// TIA Portal V20 export
DATA_BLOCK "LPFE_AdditionalAlarmData"   // DB241
TITLE = LPFE_AdditionalAlarmData
{ DB_Accessible_From_OPC_UA := 'FALSE' }
AUTHOR : DI FA SUP
FAMILY : LPFE
// Aditional information required to create the Andon and QAS Digital Events.
// stored: Access Published, DBAccessibleFromOPCUA false, DBAccessibleFromWebserver false, MemoryReserve 100, Namespace PFE
   VAR
      additionalAlarmData { ExternalAccessible := 'False'; ExternalVisible := 'False'; ExternalWritable := 'False'} : Array[0.._.CONFIGURED_ALARMS] of "LPFE_typeAdditionalAlarmData";   // Additional Alarm Data for Digital Events
   END_VAR
BEGIN
   additionalAlarmData[0].AlarmId := 3001;
   additionalAlarmData[1].AlarmId := 4001;
   additionalAlarmData[2].AlarmId := 4002;
   additionalAlarmData[3].AlarmId := 4003;
   additionalAlarmData[4].AlarmId := 4004;
   additionalAlarmData[5].AlarmId := 4006;
   additionalAlarmData[6].AlarmId := 4007;
   additionalAlarmData[7].AlarmId := 4008;
   additionalAlarmData[8].AlarmId := 4009;
   additionalAlarmData[9].AlarmId := 4010;
   additionalAlarmData[10].AlarmId := 4011;
   additionalAlarmData[11].AlarmId := 4012;
   additionalAlarmData[12].AlarmId := 4013;
   additionalAlarmData[13].AlarmId := 4014;
   additionalAlarmData[14].AlarmId := 10001;
   additionalAlarmData[15].AlarmId := 10002;
   additionalAlarmData[16].AlarmId := 10003;
   additionalAlarmData[17].AlarmId := 10004;
   additionalAlarmData[18].AlarmId := 10005;
   additionalAlarmData[19].AlarmId := 10006;
   additionalAlarmData[20].AlarmId := 10007;
   additionalAlarmData[21].AlarmId := 10008;
   additionalAlarmData[22].AlarmId := 11001;
   additionalAlarmData[23].AlarmId := 11002;
   additionalAlarmData[24].AlarmId := 11003;
   additionalAlarmData[25].AlarmId := 11004;
   additionalAlarmData[26].AlarmId := 11005;
   additionalAlarmData[27].AlarmId := 11006;
   additionalAlarmData[28].AlarmId := 11007;
   additionalAlarmData[29].AlarmId := 11008;
   additionalAlarmData[30].AlarmId := 12001;
   additionalAlarmData[31].AlarmId := 12002;
   additionalAlarmData[32].AlarmId := 12003;
   additionalAlarmData[33].AlarmId := 12004;
   additionalAlarmData[34].AlarmId := 12005;
   additionalAlarmData[35].AlarmId := 12006;
   additionalAlarmData[36].AlarmId := 12007;
   additionalAlarmData[37].AlarmId := 12008;
   additionalAlarmData[38].AlarmId := 13001;
   additionalAlarmData[39].AlarmId := 13002;
   additionalAlarmData[40].AlarmId := 13003;
   additionalAlarmData[41].AlarmId := 13004;
   additionalAlarmData[42].AlarmId := 13005;
   additionalAlarmData[43].AlarmId := 13006;
   additionalAlarmData[44].AlarmId := 13007;
   additionalAlarmData[45].AlarmId := 13008;
   additionalAlarmData[46].AlarmId := 20001;
   additionalAlarmData[47].AlarmId := 20002;
   additionalAlarmData[48].AlarmId := 20003;
   additionalAlarmData[49].AlarmId := 20004;
   additionalAlarmData[50].AlarmId := 20005;
   additionalAlarmData[51].AlarmId := 20006;
   additionalAlarmData[52].AlarmId := 20007;
   additionalAlarmData[53].AlarmId := 20008;
   additionalAlarmData[54].AlarmId := 21001;
   additionalAlarmData[55].AlarmId := 21002;
   additionalAlarmData[56].AlarmId := 21003;
   additionalAlarmData[57].AlarmId := 21004;
   additionalAlarmData[58].AlarmId := 21005;
   additionalAlarmData[59].AlarmId := 21006;
   additionalAlarmData[60].AlarmId := 21007;
   additionalAlarmData[61].AlarmId := 21008;
   additionalAlarmData[62].AlarmId := 22001;
   additionalAlarmData[63].AlarmId := 22002;
   additionalAlarmData[64].AlarmId := 22003;
   additionalAlarmData[65].AlarmId := 22004;
   additionalAlarmData[66].AlarmId := 22005;
   additionalAlarmData[67].AlarmId := 22006;
   additionalAlarmData[68].AlarmId := 22007;
   additionalAlarmData[69].AlarmId := 22008;
   additionalAlarmData[70].AlarmId := 23001;
   additionalAlarmData[71].AlarmId := 23002;
   additionalAlarmData[72].AlarmId := 23003;
   additionalAlarmData[73].AlarmId := 23004;
   additionalAlarmData[74].AlarmId := 23005;
   additionalAlarmData[75].AlarmId := 23006;
   additionalAlarmData[76].AlarmId := 23007;
   additionalAlarmData[77].AlarmId := 23008;
   additionalAlarmData[78].AlarmId := 24001;
   additionalAlarmData[79].AlarmId := 24002;
   additionalAlarmData[80].AlarmId := 24003;
   additionalAlarmData[81].AlarmId := 24004;
   additionalAlarmData[82].AlarmId := 24005;
   additionalAlarmData[83].AlarmId := 24006;
   additionalAlarmData[84].AlarmId := 24007;
   additionalAlarmData[85].AlarmId := 24008;
   additionalAlarmData[86].AlarmId := 25001;
   additionalAlarmData[87].AlarmId := 25002;
   additionalAlarmData[88].AlarmId := 25003;
   additionalAlarmData[89].AlarmId := 25004;
   additionalAlarmData[90].AlarmId := 25005;
   additionalAlarmData[91].AlarmId := 25006;
   additionalAlarmData[92].AlarmId := 25007;
   additionalAlarmData[93].AlarmId := 25008;
   additionalAlarmData[94].AlarmId := 26001;
   additionalAlarmData[95].AlarmId := 26002;
   additionalAlarmData[96].AlarmId := 26003;
   additionalAlarmData[97].AlarmId := 26004;
   additionalAlarmData[98].AlarmId := 26005;
   additionalAlarmData[99].AlarmId := 26006;
   additionalAlarmData[100].AlarmId := 26007;
   additionalAlarmData[101].AlarmId := 26008;
   additionalAlarmData[102].AlarmId := 27001;
   additionalAlarmData[103].AlarmId := 27002;
   additionalAlarmData[104].AlarmId := 27003;
   additionalAlarmData[105].AlarmId := 27004;
   additionalAlarmData[106].AlarmId := 27005;
   additionalAlarmData[107].AlarmId := 27006;
   additionalAlarmData[108].AlarmId := 27007;
   additionalAlarmData[109].AlarmId := 27008;
   additionalAlarmData[110].AlarmId := 30001;
   additionalAlarmData[111].AlarmId := 30002;
   additionalAlarmData[112].AlarmId := 30003;
   additionalAlarmData[113].AlarmId := 30004;
   additionalAlarmData[114].AlarmId := 30005;
   additionalAlarmData[115].AlarmId := 30006;
   additionalAlarmData[116].AlarmId := 30007;
   additionalAlarmData[117].AlarmId := 30008;
   additionalAlarmData[118].AlarmId := 30009;
   additionalAlarmData[119].AlarmId := 30010;
   additionalAlarmData[120].AlarmId := 30011;
   additionalAlarmData[121].AlarmId := 31001;
   additionalAlarmData[122].AlarmId := 31002;
   additionalAlarmData[123].AlarmId := 31003;
   additionalAlarmData[124].AlarmId := 31004;
   additionalAlarmData[125].AlarmId := 31005;
   additionalAlarmData[126].AlarmId := 31006;
   additionalAlarmData[127].AlarmId := 31007;
   additionalAlarmData[128].AlarmId := 31008;
   additionalAlarmData[129].AlarmId := 32001;
   additionalAlarmData[130].AlarmId := 32002;
   additionalAlarmData[131].AlarmId := 32003;
   additionalAlarmData[132].AlarmId := 32004;
   additionalAlarmData[133].AlarmId := 32005;
   additionalAlarmData[134].AlarmId := 32006;
   additionalAlarmData[135].AlarmId := 32007;
   additionalAlarmData[136].AlarmId := 32008;
   additionalAlarmData[137].AlarmId := 33001;
   additionalAlarmData[138].AlarmId := 33002;
   additionalAlarmData[139].AlarmId := 33003;
   additionalAlarmData[140].AlarmId := 33004;
   additionalAlarmData[141].AlarmId := 33005;
   additionalAlarmData[142].AlarmId := 33006;
   additionalAlarmData[143].AlarmId := 33007;
   additionalAlarmData[144].AlarmId := 33008;
   additionalAlarmData[145].AlarmId := 34001;
   additionalAlarmData[146].AlarmId := 34002;
   additionalAlarmData[147].AlarmId := 34003;
   additionalAlarmData[148].AlarmId := 34004;
   additionalAlarmData[149].AlarmId := 34005;
   additionalAlarmData[150].AlarmId := 34006;
   additionalAlarmData[151].AlarmId := 34007;
   additionalAlarmData[152].AlarmId := 34008;
   additionalAlarmData[153].AlarmId := 35001;
   additionalAlarmData[154].AlarmId := 35002;
   additionalAlarmData[155].AlarmId := 35003;
   additionalAlarmData[156].AlarmId := 35004;
   additionalAlarmData[157].AlarmId := 35005;
   additionalAlarmData[158].AlarmId := 35006;
   additionalAlarmData[159].AlarmId := 35007;
   additionalAlarmData[160].AlarmId := 35008;
   additionalAlarmData[161].AlarmId := 36001;
   additionalAlarmData[162].AlarmId := 36002;
   additionalAlarmData[163].AlarmId := 36003;
   additionalAlarmData[164].AlarmId := 36004;
   additionalAlarmData[165].AlarmId := 36005;
   additionalAlarmData[166].AlarmId := 36006;
   additionalAlarmData[167].AlarmId := 36007;
   additionalAlarmData[168].AlarmId := 36008;
   additionalAlarmData[169].AlarmId := 40001;
   additionalAlarmData[170].AlarmId := 40002;
   additionalAlarmData[171].AlarmId := 40003;
   additionalAlarmData[172].AlarmId := 40004;
   additionalAlarmData[173].AlarmId := 40005;
   additionalAlarmData[174].AlarmId := 40006;
   additionalAlarmData[175].AlarmId := 40007;
   additionalAlarmData[176].AlarmId := 40008;
   additionalAlarmData[177..999].AlarmId := 0;
   additionalAlarmData[0].priority := 15;
   additionalAlarmData[1..4].priority := 30;
   additionalAlarmData[5].priority := 151;
   additionalAlarmData[6].priority := 104;
   additionalAlarmData[7].priority := 106;
   additionalAlarmData[8].priority := 30;
   additionalAlarmData[9].priority := 151;
   additionalAlarmData[10].priority := 120;
   additionalAlarmData[11].priority := 151;
   additionalAlarmData[12].priority := 105;
   additionalAlarmData[13].priority := 151;
   additionalAlarmData[14].priority := 170;
   additionalAlarmData[15].priority := 106;
   additionalAlarmData[16].priority := 151;
   additionalAlarmData[17].priority := 152;
   additionalAlarmData[18].priority := 170;
   additionalAlarmData[19].priority := 201;
   additionalAlarmData[20].priority := 205;
   additionalAlarmData[21].priority := 251;
   additionalAlarmData[22].priority := 10;
   additionalAlarmData[23].priority := 120;
   additionalAlarmData[24].priority := 151;
   additionalAlarmData[25].priority := 152;
   additionalAlarmData[26].priority := 170;
   additionalAlarmData[27].priority := 204;
   additionalAlarmData[28].priority := 206;
   additionalAlarmData[29].priority := 254;
   additionalAlarmData[30].priority := 15;
   additionalAlarmData[31].priority := 107;
   additionalAlarmData[32].priority := 151;
   additionalAlarmData[33].priority := 152;
   additionalAlarmData[34].priority := 170;
   additionalAlarmData[35].priority := 202;
   additionalAlarmData[36].priority := 205;
   additionalAlarmData[37].priority := 251;
   additionalAlarmData[38].priority := 20;
   additionalAlarmData[39].priority := 105;
   additionalAlarmData[40].priority := 151;
   additionalAlarmData[41].priority := 152;
   additionalAlarmData[42].priority := 170;
   additionalAlarmData[43].priority := 204;
   additionalAlarmData[44].priority := 206;
   additionalAlarmData[45].priority := 251;
   additionalAlarmData[46].priority := 170;
   additionalAlarmData[47].priority := 104;
   additionalAlarmData[48].priority := 151;
   additionalAlarmData[49].priority := 152;
   additionalAlarmData[50].priority := 170;
   additionalAlarmData[51].priority := 202;
   additionalAlarmData[52].priority := 205;
   additionalAlarmData[53].priority := 251;
   additionalAlarmData[54].priority := 35;
   additionalAlarmData[55].priority := 120;
   additionalAlarmData[56].priority := 151;
   additionalAlarmData[57].priority := 152;
   additionalAlarmData[58].priority := 170;
   additionalAlarmData[59].priority := 201;
   additionalAlarmData[60].priority := 206;
   additionalAlarmData[61].priority := 254;
   additionalAlarmData[62].priority := 50;
   additionalAlarmData[63].priority := 105;
   additionalAlarmData[64].priority := 151;
   additionalAlarmData[65].priority := 152;
   additionalAlarmData[66].priority := 170;
   additionalAlarmData[67].priority := 204;
   additionalAlarmData[68].priority := 205;
   additionalAlarmData[69].priority := 254;
   additionalAlarmData[70].priority := 55;
   additionalAlarmData[71].priority := 105;
   additionalAlarmData[72].priority := 151;
   additionalAlarmData[73].priority := 152;
   additionalAlarmData[74].priority := 170;
   additionalAlarmData[75].priority := 202;
   additionalAlarmData[76].priority := 206;
   additionalAlarmData[77].priority := 251;
   additionalAlarmData[78].priority := 60;
   additionalAlarmData[79].priority := 106;
   additionalAlarmData[80].priority := 151;
   additionalAlarmData[81].priority := 152;
   additionalAlarmData[82].priority := 170;
   additionalAlarmData[83].priority := 202;
   additionalAlarmData[84].priority := 206;
   additionalAlarmData[85].priority := 254;
   additionalAlarmData[86].priority := 65;
   additionalAlarmData[87].priority := 104;
   additionalAlarmData[88].priority := 151;
   additionalAlarmData[89].priority := 152;
   additionalAlarmData[90].priority := 170;
   additionalAlarmData[91].priority := 201;
   additionalAlarmData[92].priority := 206;
   additionalAlarmData[93].priority := 251;
   additionalAlarmData[94].priority := 5;
   additionalAlarmData[95].priority := 120;
   additionalAlarmData[96].priority := 151;
   additionalAlarmData[97].priority := 152;
   additionalAlarmData[98].priority := 170;
   additionalAlarmData[99].priority := 201;
   additionalAlarmData[100].priority := 205;
   additionalAlarmData[101].priority := 251;
   additionalAlarmData[102].priority := 10;
   additionalAlarmData[103].priority := 105;
   additionalAlarmData[104].priority := 151;
   additionalAlarmData[105].priority := 152;
   additionalAlarmData[106].priority := 170;
   additionalAlarmData[107].priority := 204;
   additionalAlarmData[108].priority := 206;
   additionalAlarmData[109].priority := 254;
   additionalAlarmData[110].priority := 170;
   additionalAlarmData[111].priority := 106;
   additionalAlarmData[112].priority := 151;
   additionalAlarmData[113].priority := 152;
   additionalAlarmData[114].priority := 170;
   additionalAlarmData[115].priority := 204;
   additionalAlarmData[116].priority := 206;
   additionalAlarmData[117].priority := 251;
   additionalAlarmData[118].priority := 15;
   additionalAlarmData[119].priority := 201;
   additionalAlarmData[120].priority := 251;
   additionalAlarmData[121].priority := 10;
   additionalAlarmData[122].priority := 105;
   additionalAlarmData[123].priority := 151;
   additionalAlarmData[124].priority := 152;
   additionalAlarmData[125].priority := 170;
   additionalAlarmData[126].priority := 204;
   additionalAlarmData[127].priority := 205;
   additionalAlarmData[128].priority := 254;
   additionalAlarmData[129].priority := 35;
   additionalAlarmData[130].priority := 106;
   additionalAlarmData[131].priority := 151;
   additionalAlarmData[132].priority := 152;
   additionalAlarmData[133].priority := 170;
   additionalAlarmData[134].priority := 201;
   additionalAlarmData[135].priority := 205;
   additionalAlarmData[136].priority := 254;
   additionalAlarmData[137].priority := 30;
   additionalAlarmData[138].priority := 105;
   additionalAlarmData[139].priority := 151;
   additionalAlarmData[140].priority := 152;
   additionalAlarmData[141].priority := 170;
   additionalAlarmData[142].priority := 204;
   additionalAlarmData[143].priority := 206;
   additionalAlarmData[144].priority := 251;
   additionalAlarmData[145].priority := 65;
   additionalAlarmData[146].priority := 104;
   additionalAlarmData[147].priority := 151;
   additionalAlarmData[148].priority := 152;
   additionalAlarmData[149].priority := 170;
   additionalAlarmData[150].priority := 201;
   additionalAlarmData[151].priority := 205;
   additionalAlarmData[152].priority := 254;
   additionalAlarmData[153].priority := 60;
   additionalAlarmData[154].priority := 105;
   additionalAlarmData[155].priority := 151;
   additionalAlarmData[156].priority := 152;
   additionalAlarmData[157].priority := 170;
   additionalAlarmData[158].priority := 201;
   additionalAlarmData[159].priority := 206;
   additionalAlarmData[160].priority := 251;
   additionalAlarmData[161].priority := 90;
   additionalAlarmData[162].priority := 120;
   additionalAlarmData[163].priority := 151;
   additionalAlarmData[164].priority := 152;
   additionalAlarmData[165].priority := 170;
   additionalAlarmData[166].priority := 204;
   additionalAlarmData[167].priority := 206;
   additionalAlarmData[168].priority := 254;
   additionalAlarmData[169].priority := 170;
   additionalAlarmData[170].priority := 104;
   additionalAlarmData[171].priority := 151;
   additionalAlarmData[172].priority := 152;
   additionalAlarmData[173].priority := 170;
   additionalAlarmData[174].priority := 204;
   additionalAlarmData[175].priority := 205;
   additionalAlarmData[176].priority := 251;
   additionalAlarmData[177..999].priority := 0;
   additionalAlarmData[0..45].CellID := 1;
   additionalAlarmData[46..109].CellID := 2;
   additionalAlarmData[110..168].CellID := 3;
   additionalAlarmData[169..176].CellID := 4;
   additionalAlarmData[177..999].CellID := 0;
   additionalAlarmData[0].subType := 150;
   additionalAlarmData[1].subType := 0;
   additionalAlarmData[2].subType := 150;
   additionalAlarmData[3].subType := 0;
   additionalAlarmData[4].subType := 150;
   additionalAlarmData[5].subType := 0;
   additionalAlarmData[6].subType := 150;
   additionalAlarmData[7].subType := 0;
   additionalAlarmData[8].subType := 150;
   additionalAlarmData[9].subType := 0;
   additionalAlarmData[10].subType := 150;
   additionalAlarmData[11].subType := 0;
   additionalAlarmData[12].subType := 150;
   additionalAlarmData[13].subType := 0;
   additionalAlarmData[14].subType := 150;
   additionalAlarmData[15].subType := 0;
   additionalAlarmData[16].subType := 150;
   additionalAlarmData[17].subType := 0;
   additionalAlarmData[18].subType := 150;
   additionalAlarmData[19].subType := 0;
   additionalAlarmData[20].subType := 150;
   additionalAlarmData[21].subType := 0;
   additionalAlarmData[22].subType := 150;
   additionalAlarmData[23].subType := 0;
   additionalAlarmData[24].subType := 150;
   additionalAlarmData[25].subType := 0;
   additionalAlarmData[26].subType := 150;
   additionalAlarmData[27].subType := 0;
   additionalAlarmData[28].subType := 150;
   additionalAlarmData[29].subType := 0;
   additionalAlarmData[30].subType := 150;
   additionalAlarmData[31].subType := 0;
   additionalAlarmData[32].subType := 150;
   additionalAlarmData[33].subType := 0;
   additionalAlarmData[34].subType := 150;
   additionalAlarmData[35].subType := 0;
   additionalAlarmData[36].subType := 150;
   additionalAlarmData[37].subType := 0;
   additionalAlarmData[38].subType := 150;
   additionalAlarmData[39].subType := 0;
   additionalAlarmData[40].subType := 150;
   additionalAlarmData[41].subType := 0;
   additionalAlarmData[42].subType := 150;
   additionalAlarmData[43].subType := 0;
   additionalAlarmData[44].subType := 150;
   additionalAlarmData[45].subType := 0;
   additionalAlarmData[46].subType := 150;
   additionalAlarmData[47].subType := 0;
   additionalAlarmData[48].subType := 150;
   additionalAlarmData[49].subType := 0;
   additionalAlarmData[50].subType := 150;
   additionalAlarmData[51].subType := 0;
   additionalAlarmData[52].subType := 150;
   additionalAlarmData[53].subType := 0;
   additionalAlarmData[54].subType := 150;
   additionalAlarmData[55].subType := 0;
   additionalAlarmData[56].subType := 150;
   additionalAlarmData[57].subType := 0;
   additionalAlarmData[58].subType := 150;
   additionalAlarmData[59].subType := 0;
   additionalAlarmData[60].subType := 150;
   additionalAlarmData[61].subType := 0;
   additionalAlarmData[62..63].subType := 150;
   additionalAlarmData[64].subType := 0;
   additionalAlarmData[65].subType := 150;
   additionalAlarmData[66].subType := 0;
   additionalAlarmData[67].subType := 150;
   additionalAlarmData[68].subType := 0;
   additionalAlarmData[69].subType := 150;
   additionalAlarmData[70].subType := 0;
   additionalAlarmData[71].subType := 150;
   additionalAlarmData[72].subType := 0;
   additionalAlarmData[73].subType := 150;
   additionalAlarmData[74].subType := 0;
   additionalAlarmData[75].subType := 150;
   additionalAlarmData[76].subType := 0;
   additionalAlarmData[77].subType := 150;
   additionalAlarmData[78].subType := 0;
   additionalAlarmData[79].subType := 150;
   additionalAlarmData[80].subType := 0;
   additionalAlarmData[81].subType := 150;
   additionalAlarmData[82].subType := 0;
   additionalAlarmData[83].subType := 150;
   additionalAlarmData[84].subType := 0;
   additionalAlarmData[85].subType := 150;
   additionalAlarmData[86].subType := 0;
   additionalAlarmData[87].subType := 150;
   additionalAlarmData[88].subType := 0;
   additionalAlarmData[89].subType := 150;
   additionalAlarmData[90].subType := 0;
   additionalAlarmData[91].subType := 150;
   additionalAlarmData[92].subType := 0;
   additionalAlarmData[93].subType := 150;
   additionalAlarmData[94].subType := 0;
   additionalAlarmData[95].subType := 150;
   additionalAlarmData[96].subType := 0;
   additionalAlarmData[97].subType := 150;
   additionalAlarmData[98].subType := 0;
   additionalAlarmData[99].subType := 150;
   additionalAlarmData[100].subType := 0;
   additionalAlarmData[101].subType := 150;
   additionalAlarmData[102].subType := 0;
   additionalAlarmData[103].subType := 150;
   additionalAlarmData[104].subType := 0;
   additionalAlarmData[105].subType := 150;
   additionalAlarmData[106].subType := 0;
   additionalAlarmData[107].subType := 150;
   additionalAlarmData[108].subType := 0;
   additionalAlarmData[109..110].subType := 150;
   additionalAlarmData[111].subType := 0;
   additionalAlarmData[112].subType := 150;
   additionalAlarmData[113].subType := 0;
   additionalAlarmData[114].subType := 150;
   additionalAlarmData[115].subType := 0;
   additionalAlarmData[116].subType := 150;
   additionalAlarmData[117].subType := 0;
   additionalAlarmData[118..119].subType := 150;
   additionalAlarmData[120].subType := 0;
   additionalAlarmData[121].subType := 150;
   additionalAlarmData[122].subType := 0;
   additionalAlarmData[123].subType := 150;
   additionalAlarmData[124].subType := 0;
   additionalAlarmData[125..126].subType := 150;
   additionalAlarmData[127].subType := 0;
   additionalAlarmData[128].subType := 150;
   additionalAlarmData[129].subType := 0;
   additionalAlarmData[130..131].subType := 150;
   additionalAlarmData[132].subType := 0;
   additionalAlarmData[133].subType := 150;
   additionalAlarmData[134].subType := 0;
   additionalAlarmData[135].subType := 150;
   additionalAlarmData[136].subType := 0;
   additionalAlarmData[137].subType := 150;
   additionalAlarmData[138].subType := 0;
   additionalAlarmData[139].subType := 150;
   additionalAlarmData[140].subType := 0;
   additionalAlarmData[141].subType := 150;
   additionalAlarmData[142].subType := 0;
   additionalAlarmData[143].subType := 150;
   additionalAlarmData[144..145].subType := 0;
   additionalAlarmData[146..148].subType := 150;
   additionalAlarmData[149].subType := 0;
   additionalAlarmData[150].subType := 150;
   additionalAlarmData[151].subType := 0;
   additionalAlarmData[152].subType := 150;
   additionalAlarmData[153].subType := 0;
   additionalAlarmData[154].subType := 150;
   additionalAlarmData[155].subType := 0;
   additionalAlarmData[156].subType := 150;
   additionalAlarmData[157].subType := 0;
   additionalAlarmData[158].subType := 150;
   additionalAlarmData[159].subType := 0;
   additionalAlarmData[160].subType := 150;
   additionalAlarmData[161].subType := 0;
   additionalAlarmData[162].subType := 150;
   additionalAlarmData[163].subType := 0;
   additionalAlarmData[164].subType := 150;
   additionalAlarmData[165..166].subType := 0;
   additionalAlarmData[167].subType := 150;
   additionalAlarmData[168].subType := 0;
   additionalAlarmData[169].subType := 150;
   additionalAlarmData[170].subType := 0;
   additionalAlarmData[171].subType := 150;
   additionalAlarmData[172..173].subType := 0;
   additionalAlarmData[174].subType := 150;
   additionalAlarmData[175].subType := 0;
   additionalAlarmData[176].subType := 150;
   additionalAlarmData[177..999].subType := 0;
   additionalAlarmData[0].classification[0] := 'M';
   additionalAlarmData[0].classification[1] := 'F';
   additionalAlarmData[0].classification[2..3] := ' ';
   additionalAlarmData[1].classification[0] := 'M';
   additionalAlarmData[1].classification[1] := 'F';
   additionalAlarmData[1].classification[2..3] := ' ';
   additionalAlarmData[2].classification[0] := 'M';
   additionalAlarmData[2].classification[1] := 'F';
   additionalAlarmData[2].classification[2..3] := ' ';
   additionalAlarmData[3].classification[0] := 'M';
   additionalAlarmData[3].classification[1] := 'F';
   additionalAlarmData[3].classification[2..3] := ' ';
   additionalAlarmData[4].classification[0] := 'M';
   additionalAlarmData[4].classification[1] := 'F';
   additionalAlarmData[4].classification[2..3] := ' ';
   additionalAlarmData[5].classification[0] := 'T';
   additionalAlarmData[5].classification[1] := 'F';
   additionalAlarmData[5].classification[2] := 'I';
   additionalAlarmData[5].classification[3] := 'B';
   additionalAlarmData[6].classification[0] := 'P';
   additionalAlarmData[6].classification[1] := 'F';
   additionalAlarmData[6].classification[2..3] := ' ';
   additionalAlarmData[7].classification[0] := 'P';
   additionalAlarmData[7].classification[1] := 'F';
   additionalAlarmData[7].classification[2..3] := ' ';
   additionalAlarmData[8].classification[0] := 'M';
   additionalAlarmData[8].classification[1] := 'F';
   additionalAlarmData[8].classification[2..3] := ' ';
   additionalAlarmData[9].classification[0] := 'T';
   additionalAlarmData[9].classification[1] := 'F';
   additionalAlarmData[9].classification[2] := 'I';
   additionalAlarmData[9].classification[3] := 'B';
   additionalAlarmData[10].classification[0] := 'P';
   additionalAlarmData[10].classification[1] := 'F';
   additionalAlarmData[10].classification[2..3] := ' ';
   additionalAlarmData[11].classification[0] := 'T';
   additionalAlarmData[11].classification[1] := 'F';
   additionalAlarmData[11].classification[2] := 'I';
   additionalAlarmData[11].classification[3] := 'B';
   additionalAlarmData[12].classification[0] := 'P';
   additionalAlarmData[12].classification[1] := 'F';
   additionalAlarmData[12].classification[2..3] := ' ';
   additionalAlarmData[13].classification[0] := 'T';
   additionalAlarmData[13].classification[1] := 'F';
   additionalAlarmData[13].classification[2] := 'I';
   additionalAlarmData[13].classification[3] := 'B';
   additionalAlarmData[14].classification[0] := 'S';
   additionalAlarmData[14].classification[1] := 'F';
   additionalAlarmData[14].classification[2..3] := ' ';
   additionalAlarmData[15].classification[0] := 'P';
   additionalAlarmData[15].classification[1] := 'F';
   additionalAlarmData[15].classification[2..3] := ' ';
   additionalAlarmData[16].classification[0] := 'T';
   additionalAlarmData[16].classification[1] := 'F';
   additionalAlarmData[16].classification[2] := 'I';
   additionalAlarmData[16].classification[3] := 'B';
   additionalAlarmData[17].classification[0] := 'T';
   additionalAlarmData[17].classification[1] := 'F';
   additionalAlarmData[17].classification[2] := 'S';
   additionalAlarmData[17].classification[3] := ' ';
   additionalAlarmData[18].classification[0] := 'S';
   additionalAlarmData[18].classification[1] := 'F';
   additionalAlarmData[18].classification[2..3] := ' ';
   additionalAlarmData[19].classification[0] := 'M';
   additionalAlarmData[19].classification[1] := 'W';
   additionalAlarmData[19].classification[2..3] := ' ';
   additionalAlarmData[20].classification[0] := 'P';
   additionalAlarmData[20].classification[1] := 'W';
   additionalAlarmData[20].classification[2..3] := ' ';
   additionalAlarmData[21].classification[0] := 'M';
   additionalAlarmData[21].classification[1] := 'S';
   additionalAlarmData[21].classification[2..3] := ' ';
   additionalAlarmData[22].classification[0] := 'M';
   additionalAlarmData[22].classification[1] := 'F';
   additionalAlarmData[22].classification[2..3] := ' ';
   additionalAlarmData[23].classification[0] := 'P';
   additionalAlarmData[23].classification[1] := 'F';
   additionalAlarmData[23].classification[2..3] := ' ';
   additionalAlarmData[24].classification[0] := 'T';
   additionalAlarmData[24].classification[1] := 'F';
   additionalAlarmData[24].classification[2] := 'I';
   additionalAlarmData[24].classification[3] := 'B';
   additionalAlarmData[25].classification[0] := 'T';
   additionalAlarmData[25].classification[1] := 'F';
   additionalAlarmData[25].classification[2] := 'S';
   additionalAlarmData[25].classification[3] := ' ';
   additionalAlarmData[26].classification[0] := 'S';
   additionalAlarmData[26].classification[1] := 'F';
   additionalAlarmData[26].classification[2..3] := ' ';
   additionalAlarmData[27].classification[0] := 'M';
   additionalAlarmData[27].classification[1] := 'W';
   additionalAlarmData[27].classification[2..3] := ' ';
   additionalAlarmData[28].classification[0] := 'P';
   additionalAlarmData[28].classification[1] := 'W';
   additionalAlarmData[28].classification[2..3] := ' ';
   additionalAlarmData[29].classification[0] := 'M';
   additionalAlarmData[29].classification[1] := 'S';
   additionalAlarmData[29].classification[2..3] := ' ';
   additionalAlarmData[30].classification[0] := 'M';
   additionalAlarmData[30].classification[1] := 'F';
   additionalAlarmData[30].classification[2..3] := ' ';
   additionalAlarmData[31].classification[0] := 'P';
   additionalAlarmData[31].classification[1] := 'F';
   additionalAlarmData[31].classification[2..3] := ' ';
   additionalAlarmData[32].classification[0] := 'T';
   additionalAlarmData[32].classification[1] := 'F';
   additionalAlarmData[32].classification[2] := 'I';
   additionalAlarmData[32].classification[3] := 'B';
   additionalAlarmData[33].classification[0] := 'T';
   additionalAlarmData[33].classification[1] := 'F';
   additionalAlarmData[33].classification[2] := 'S';
   additionalAlarmData[33].classification[3] := ' ';
   additionalAlarmData[34].classification[0] := 'S';
   additionalAlarmData[34].classification[1] := 'F';
   additionalAlarmData[34].classification[2..3] := ' ';
   additionalAlarmData[35].classification[0] := 'M';
   additionalAlarmData[35].classification[1] := 'W';
   additionalAlarmData[35].classification[2..3] := ' ';
   additionalAlarmData[36].classification[0] := 'P';
   additionalAlarmData[36].classification[1] := 'W';
   additionalAlarmData[36].classification[2..3] := ' ';
   additionalAlarmData[37].classification[0] := 'M';
   additionalAlarmData[37].classification[1] := 'S';
   additionalAlarmData[37].classification[2..3] := ' ';
   additionalAlarmData[38].classification[0] := 'M';
   additionalAlarmData[38].classification[1] := 'F';
   additionalAlarmData[38].classification[2..3] := ' ';
   additionalAlarmData[39].classification[0] := 'P';
   additionalAlarmData[39].classification[1] := 'F';
   additionalAlarmData[39].classification[2..3] := ' ';
   additionalAlarmData[40].classification[0] := 'T';
   additionalAlarmData[40].classification[1] := 'F';
   additionalAlarmData[40].classification[2] := 'I';
   additionalAlarmData[40].classification[3] := 'B';
   additionalAlarmData[41].classification[0] := 'T';
   additionalAlarmData[41].classification[1] := 'F';
   additionalAlarmData[41].classification[2] := 'S';
   additionalAlarmData[41].classification[3] := ' ';
   additionalAlarmData[42].classification[0] := 'S';
   additionalAlarmData[42].classification[1] := 'F';
   additionalAlarmData[42].classification[2..3] := ' ';
   additionalAlarmData[43].classification[0] := 'M';
   additionalAlarmData[43].classification[1] := 'W';
   additionalAlarmData[43].classification[2..3] := ' ';
   additionalAlarmData[44].classification[0] := 'P';
   additionalAlarmData[44].classification[1] := 'W';
   additionalAlarmData[44].classification[2..3] := ' ';
   additionalAlarmData[45].classification[0] := 'M';
   additionalAlarmData[45].classification[1] := 'S';
   additionalAlarmData[45].classification[2..3] := ' ';
   additionalAlarmData[46].classification[0] := 'S';
   additionalAlarmData[46].classification[1] := 'F';
   additionalAlarmData[46].classification[2..3] := ' ';
   additionalAlarmData[47].classification[0] := 'P';
   additionalAlarmData[47].classification[1] := 'F';
   additionalAlarmData[47].classification[2..3] := ' ';
   additionalAlarmData[48].classification[0] := 'T';
   additionalAlarmData[48].classification[1] := 'F';
   additionalAlarmData[48].classification[2] := 'I';
   additionalAlarmData[48].classification[3] := 'B';
   additionalAlarmData[49].classification[0] := 'T';
   additionalAlarmData[49].classification[1] := 'F';
   additionalAlarmData[49].classification[2] := 'S';
   additionalAlarmData[49].classification[3] := ' ';
   additionalAlarmData[50].classification[0] := 'S';
   additionalAlarmData[50].classification[1] := 'F';
   additionalAlarmData[50].classification[2..3] := ' ';
   additionalAlarmData[51].classification[0] := 'M';
   additionalAlarmData[51].classification[1] := 'W';
   additionalAlarmData[51].classification[2..3] := ' ';
   additionalAlarmData[52].classification[0] := 'P';
   additionalAlarmData[52].classification[1] := 'W';
   additionalAlarmData[52].classification[2..3] := ' ';
   additionalAlarmData[53].classification[0] := 'M';
   additionalAlarmData[53].classification[1] := 'S';
   additionalAlarmData[53].classification[2..3] := ' ';
   additionalAlarmData[54].classification[0] := 'M';
   additionalAlarmData[54].classification[1] := 'F';
   additionalAlarmData[54].classification[2..3] := ' ';
   additionalAlarmData[55].classification[0] := 'P';
   additionalAlarmData[55].classification[1] := 'F';
   additionalAlarmData[55].classification[2..3] := ' ';
   additionalAlarmData[56].classification[0] := 'T';
   additionalAlarmData[56].classification[1] := 'F';
   additionalAlarmData[56].classification[2] := 'I';
   additionalAlarmData[56].classification[3] := 'B';
   additionalAlarmData[57].classification[0] := 'T';
   additionalAlarmData[57].classification[1] := 'F';
   additionalAlarmData[57].classification[2] := 'S';
   additionalAlarmData[57].classification[3] := ' ';
   additionalAlarmData[58].classification[0] := 'S';
   additionalAlarmData[58].classification[1] := 'F';
   additionalAlarmData[58].classification[2..3] := ' ';
   additionalAlarmData[59].classification[0] := 'M';
   additionalAlarmData[59].classification[1] := 'W';
   additionalAlarmData[59].classification[2..3] := ' ';
   additionalAlarmData[60].classification[0] := 'P';
   additionalAlarmData[60].classification[1] := 'W';
   additionalAlarmData[60].classification[2..3] := ' ';
   additionalAlarmData[61].classification[0] := 'M';
   additionalAlarmData[61].classification[1] := 'S';
   additionalAlarmData[61].classification[2..3] := ' ';
   additionalAlarmData[62].classification[0] := 'M';
   additionalAlarmData[62].classification[1] := 'F';
   additionalAlarmData[62].classification[2..3] := ' ';
   additionalAlarmData[63].classification[0] := 'P';
   additionalAlarmData[63].classification[1] := 'F';
   additionalAlarmData[63].classification[2..3] := ' ';
   additionalAlarmData[64].classification[0] := 'T';
   additionalAlarmData[64].classification[1] := 'F';
   additionalAlarmData[64].classification[2] := 'I';
   additionalAlarmData[64].classification[3] := 'B';
   additionalAlarmData[65].classification[0] := 'T';
   additionalAlarmData[65].classification[1] := 'F';
   additionalAlarmData[65].classification[2] := 'S';
   additionalAlarmData[65].classification[3] := ' ';
   additionalAlarmData[66].classification[0] := 'S';
   additionalAlarmData[66].classification[1] := 'F';
   additionalAlarmData[66].classification[2..3] := ' ';
   additionalAlarmData[67].classification[0] := 'M';
   additionalAlarmData[67].classification[1] := 'W';
   additionalAlarmData[67].classification[2..3] := ' ';
   additionalAlarmData[68].classification[0] := 'P';
   additionalAlarmData[68].classification[1] := 'W';
   additionalAlarmData[68].classification[2..3] := ' ';
   additionalAlarmData[69].classification[0] := 'M';
   additionalAlarmData[69].classification[1] := 'S';
   additionalAlarmData[69].classification[2..3] := ' ';
   additionalAlarmData[70].classification[0] := 'M';
   additionalAlarmData[70].classification[1] := 'F';
   additionalAlarmData[70].classification[2..3] := ' ';
   additionalAlarmData[71].classification[0] := 'P';
   additionalAlarmData[71].classification[1] := 'F';
   additionalAlarmData[71].classification[2..3] := ' ';
   additionalAlarmData[72].classification[0] := 'T';
   additionalAlarmData[72].classification[1] := 'F';
   additionalAlarmData[72].classification[2] := 'I';
   additionalAlarmData[72].classification[3] := 'B';
   additionalAlarmData[73].classification[0] := 'T';
   additionalAlarmData[73].classification[1] := 'F';
   additionalAlarmData[73].classification[2] := 'S';
   additionalAlarmData[73].classification[3] := ' ';
   additionalAlarmData[74].classification[0] := 'S';
   additionalAlarmData[74].classification[1] := 'F';
   additionalAlarmData[74].classification[2..3] := ' ';
   additionalAlarmData[75].classification[0] := 'M';
   additionalAlarmData[75].classification[1] := 'W';
   additionalAlarmData[75].classification[2..3] := ' ';
   additionalAlarmData[76].classification[0] := 'P';
   additionalAlarmData[76].classification[1] := 'W';
   additionalAlarmData[76].classification[2..3] := ' ';
   additionalAlarmData[77].classification[0] := 'M';
   additionalAlarmData[77].classification[1] := 'S';
   additionalAlarmData[77].classification[2..3] := ' ';
   additionalAlarmData[78].classification[0] := 'M';
   additionalAlarmData[78].classification[1] := 'F';
   additionalAlarmData[78].classification[2..3] := ' ';
   additionalAlarmData[79].classification[0] := 'P';
   additionalAlarmData[79].classification[1] := 'F';
   additionalAlarmData[79].classification[2..3] := ' ';
   additionalAlarmData[80].classification[0] := 'T';
   additionalAlarmData[80].classification[1] := 'F';
   additionalAlarmData[80].classification[2] := 'I';
   additionalAlarmData[80].classification[3] := 'B';
   additionalAlarmData[81].classification[0] := 'T';
   additionalAlarmData[81].classification[1] := 'F';
   additionalAlarmData[81].classification[2] := 'S';
   additionalAlarmData[81].classification[3] := ' ';
   additionalAlarmData[82].classification[0] := 'S';
   additionalAlarmData[82].classification[1] := 'F';
   additionalAlarmData[82].classification[2..3] := ' ';
   additionalAlarmData[83].classification[0] := 'M';
   additionalAlarmData[83].classification[1] := 'W';
   additionalAlarmData[83].classification[2..3] := ' ';
   additionalAlarmData[84].classification[0] := 'P';
   additionalAlarmData[84].classification[1] := 'W';
   additionalAlarmData[84].classification[2..3] := ' ';
   additionalAlarmData[85].classification[0] := 'M';
   additionalAlarmData[85].classification[1] := 'S';
   additionalAlarmData[85].classification[2..3] := ' ';
   additionalAlarmData[86].classification[0] := 'M';
   additionalAlarmData[86].classification[1] := 'F';
   additionalAlarmData[86].classification[2..3] := ' ';
   additionalAlarmData[87].classification[0] := 'P';
   additionalAlarmData[87].classification[1] := 'F';
   additionalAlarmData[87].classification[2..3] := ' ';
   additionalAlarmData[88].classification[0] := 'T';
   additionalAlarmData[88].classification[1] := 'F';
   additionalAlarmData[88].classification[2] := 'I';
   additionalAlarmData[88].classification[3] := 'B';
   additionalAlarmData[89].classification[0] := 'T';
   additionalAlarmData[89].classification[1] := 'F';
   additionalAlarmData[89].classification[2] := 'S';
   additionalAlarmData[89].classification[3] := ' ';
   additionalAlarmData[90].classification[0] := 'S';
   additionalAlarmData[90].classification[1] := 'F';
   additionalAlarmData[90].classification[2..3] := ' ';
   additionalAlarmData[91].classification[0] := 'M';
   additionalAlarmData[91].classification[1] := 'W';
   additionalAlarmData[91].classification[2..3] := ' ';
   additionalAlarmData[92].classification[0] := 'P';
   additionalAlarmData[92].classification[1] := 'W';
   additionalAlarmData[92].classification[2..3] := ' ';
   additionalAlarmData[93].classification[0] := 'M';
   additionalAlarmData[93].classification[1] := 'S';
   additionalAlarmData[93].classification[2..3] := ' ';
   additionalAlarmData[94].classification[0] := 'M';
   additionalAlarmData[94].classification[1] := 'F';
   additionalAlarmData[94].classification[2..3] := ' ';
   additionalAlarmData[95].classification[0] := 'P';
   additionalAlarmData[95].classification[1] := 'F';
   additionalAlarmData[95].classification[2..3] := ' ';
   additionalAlarmData[96].classification[0] := 'T';
   additionalAlarmData[96].classification[1] := 'F';
   additionalAlarmData[96].classification[2] := 'I';
   additionalAlarmData[96].classification[3] := 'B';
   additionalAlarmData[97].classification[0] := 'T';
   additionalAlarmData[97].classification[1] := 'F';
   additionalAlarmData[97].classification[2] := 'S';
   additionalAlarmData[97].classification[3] := ' ';
   additionalAlarmData[98].classification[0] := 'S';
   additionalAlarmData[98].classification[1] := 'F';
   additionalAlarmData[98].classification[2..3] := ' ';
   additionalAlarmData[99].classification[0] := 'M';
   additionalAlarmData[99].classification[1] := 'W';
   additionalAlarmData[99].classification[2..3] := ' ';
   additionalAlarmData[100].classification[0] := 'P';
   additionalAlarmData[100].classification[1] := 'W';
   additionalAlarmData[100].classification[2..3] := ' ';
   additionalAlarmData[101].classification[0] := 'M';
   additionalAlarmData[101].classification[1] := 'S';
   additionalAlarmData[101].classification[2..3] := ' ';
   additionalAlarmData[102].classification[0] := 'M';
   additionalAlarmData[102].classification[1] := 'F';
   additionalAlarmData[102].classification[2..3] := ' ';
   additionalAlarmData[103].classification[0] := 'P';
   additionalAlarmData[103].classification[1] := 'F';
   additionalAlarmData[103].classification[2..3] := ' ';
   additionalAlarmData[104].classification[0] := 'T';
   additionalAlarmData[104].classification[1] := 'F';
   additionalAlarmData[104].classification[2] := 'I';
   additionalAlarmData[104].classification[3] := 'B';
   additionalAlarmData[105].classification[0] := 'T';
   additionalAlarmData[105].classification[1] := 'F';
   additionalAlarmData[105].classification[2] := 'S';
   additionalAlarmData[105].classification[3] := ' ';
   additionalAlarmData[106].classification[0] := 'S';
   additionalAlarmData[106].classification[1] := 'F';
   additionalAlarmData[106].classification[2..3] := ' ';
   additionalAlarmData[107].classification[0] := 'M';
   additionalAlarmData[107].classification[1] := 'W';
   additionalAlarmData[107].classification[2..3] := ' ';
   additionalAlarmData[108].classification[0] := 'P';
   additionalAlarmData[108].classification[1] := 'W';
   additionalAlarmData[108].classification[2..3] := ' ';
   additionalAlarmData[109].classification[0] := 'M';
   additionalAlarmData[109].classification[1] := 'S';
   additionalAlarmData[109].classification[2..3] := ' ';
   additionalAlarmData[110].classification[0] := 'S';
   additionalAlarmData[110].classification[1] := 'F';
   additionalAlarmData[110].classification[2..3] := ' ';
   additionalAlarmData[111].classification[0] := 'P';
   additionalAlarmData[111].classification[1] := 'F';
   additionalAlarmData[111].classification[2..3] := ' ';
   additionalAlarmData[112].classification[0] := 'T';
   additionalAlarmData[112].classification[1] := 'F';
   additionalAlarmData[112].classification[2] := 'I';
   additionalAlarmData[112].classification[3] := 'B';
   additionalAlarmData[113].classification[0] := 'T';
   additionalAlarmData[113].classification[1] := 'F';
   additionalAlarmData[113].classification[2] := 'S';
   additionalAlarmData[113].classification[3] := ' ';
   additionalAlarmData[114].classification[0] := 'S';
   additionalAlarmData[114].classification[1] := 'F';
   additionalAlarmData[114].classification[2..3] := ' ';
   additionalAlarmData[115].classification[0] := 'M';
   additionalAlarmData[115].classification[1] := 'W';
   additionalAlarmData[115].classification[2..3] := ' ';
   additionalAlarmData[116].classification[0] := 'P';
   additionalAlarmData[116].classification[1] := 'W';
   additionalAlarmData[116].classification[2..3] := ' ';
   additionalAlarmData[117].classification[0] := 'M';
   additionalAlarmData[117].classification[1] := 'S';
   additionalAlarmData[117].classification[2..3] := ' ';
   additionalAlarmData[118].classification[0] := 'M';
   additionalAlarmData[118].classification[1] := 'F';
   additionalAlarmData[118].classification[2..3] := ' ';
   additionalAlarmData[119].classification[0] := 'M';
   additionalAlarmData[119].classification[1] := 'W';
   additionalAlarmData[119].classification[2..3] := ' ';
   additionalAlarmData[120].classification[0] := 'M';
   additionalAlarmData[120].classification[1] := 'S';
   additionalAlarmData[120].classification[2..3] := ' ';
   additionalAlarmData[121].classification[0] := 'M';
   additionalAlarmData[121].classification[1] := 'F';
   additionalAlarmData[121].classification[2..3] := ' ';
   additionalAlarmData[122].classification[0] := 'P';
   additionalAlarmData[122].classification[1] := 'F';
   additionalAlarmData[122].classification[2..3] := ' ';
   additionalAlarmData[123].classification[0] := 'T';
   additionalAlarmData[123].classification[1] := 'F';
   additionalAlarmData[123].classification[2] := 'I';
   additionalAlarmData[123].classification[3] := 'B';
   additionalAlarmData[124].classification[0] := 'T';
   additionalAlarmData[124].classification[1] := 'F';
   additionalAlarmData[124].classification[2] := 'S';
   additionalAlarmData[124].classification[3] := ' ';
   additionalAlarmData[125].classification[0] := 'S';
   additionalAlarmData[125].classification[1] := 'F';
   additionalAlarmData[125].classification[2..3] := ' ';
   additionalAlarmData[126].classification[0] := 'M';
   additionalAlarmData[126].classification[1] := 'W';
   additionalAlarmData[126].classification[2..3] := ' ';
   additionalAlarmData[127].classification[0] := 'P';
   additionalAlarmData[127].classification[1] := 'W';
   additionalAlarmData[127].classification[2..3] := ' ';
   additionalAlarmData[128].classification[0] := 'M';
   additionalAlarmData[128].classification[1] := 'S';
   additionalAlarmData[128].classification[2..3] := ' ';
   additionalAlarmData[129].classification[0] := 'M';
   additionalAlarmData[129].classification[1] := 'F';
   additionalAlarmData[129].classification[2..3] := ' ';
   additionalAlarmData[130].classification[0] := 'P';
   additionalAlarmData[130].classification[1] := 'F';
   additionalAlarmData[130].classification[2..3] := ' ';
   additionalAlarmData[131].classification[0] := 'T';
   additionalAlarmData[131].classification[1] := 'F';
   additionalAlarmData[131].classification[2] := 'I';
   additionalAlarmData[131].classification[3] := 'B';
   additionalAlarmData[132].classification[0] := 'T';
   additionalAlarmData[132].classification[1] := 'F';
   additionalAlarmData[132].classification[2] := 'S';
   additionalAlarmData[132].classification[3] := ' ';
   additionalAlarmData[133].classification[0] := 'S';
   additionalAlarmData[133].classification[1] := 'F';
   additionalAlarmData[133].classification[2..3] := ' ';
   additionalAlarmData[134].classification[0] := 'M';
   additionalAlarmData[134].classification[1] := 'W';
   additionalAlarmData[134].classification[2..3] := ' ';
   additionalAlarmData[135].classification[0] := 'P';
   additionalAlarmData[135].classification[1] := 'W';
   additionalAlarmData[135].classification[2..3] := ' ';
   additionalAlarmData[136].classification[0] := 'M';
   additionalAlarmData[136].classification[1] := 'S';
   additionalAlarmData[136].classification[2..3] := ' ';
   additionalAlarmData[137].classification[0] := 'M';
   additionalAlarmData[137].classification[1] := 'F';
   additionalAlarmData[137].classification[2..3] := ' ';
   additionalAlarmData[138].classification[0] := 'P';
   additionalAlarmData[138].classification[1] := 'F';
   additionalAlarmData[138].classification[2..3] := ' ';
   additionalAlarmData[139].classification[0] := 'T';
   additionalAlarmData[139].classification[1] := 'F';
   additionalAlarmData[139].classification[2] := 'I';
   additionalAlarmData[139].classification[3] := 'B';
   additionalAlarmData[140].classification[0] := 'T';
   additionalAlarmData[140].classification[1] := 'F';
   additionalAlarmData[140].classification[2] := 'S';
   additionalAlarmData[140].classification[3] := ' ';
   additionalAlarmData[141].classification[0] := 'S';
   additionalAlarmData[141].classification[1] := 'F';
   additionalAlarmData[141].classification[2..3] := ' ';
   additionalAlarmData[142].classification[0] := 'M';
   additionalAlarmData[142].classification[1] := 'W';
   additionalAlarmData[142].classification[2..3] := ' ';
   additionalAlarmData[143].classification[0] := 'P';
   additionalAlarmData[143].classification[1] := 'W';
   additionalAlarmData[143].classification[2..3] := ' ';
   additionalAlarmData[144].classification[0] := 'M';
   additionalAlarmData[144].classification[1] := 'S';
   additionalAlarmData[144].classification[2..3] := ' ';
   additionalAlarmData[145].classification[0] := 'M';
   additionalAlarmData[145].classification[1] := 'F';
   additionalAlarmData[145].classification[2..3] := ' ';
   additionalAlarmData[146].classification[0] := 'P';
   additionalAlarmData[146].classification[1] := 'F';
   additionalAlarmData[146].classification[2..3] := ' ';
   additionalAlarmData[147].classification[0] := 'T';
   additionalAlarmData[147].classification[1] := 'F';
   additionalAlarmData[147].classification[2] := 'I';
   additionalAlarmData[147].classification[3] := 'B';
   additionalAlarmData[148].classification[0] := 'T';
   additionalAlarmData[148].classification[1] := 'F';
   additionalAlarmData[148].classification[2] := 'S';
   additionalAlarmData[148].classification[3] := ' ';
   additionalAlarmData[149].classification[0] := 'S';
   additionalAlarmData[149].classification[1] := 'F';
   additionalAlarmData[149].classification[2..3] := ' ';
   additionalAlarmData[150].classification[0] := 'M';
   additionalAlarmData[150].classification[1] := 'W';
   additionalAlarmData[150].classification[2..3] := ' ';
   additionalAlarmData[151].classification[0] := 'P';
   additionalAlarmData[151].classification[1] := 'W';
   additionalAlarmData[151].classification[2..3] := ' ';
   additionalAlarmData[152].classification[0] := 'M';
   additionalAlarmData[152].classification[1] := 'S';
   additionalAlarmData[152].classification[2..3] := ' ';
   additionalAlarmData[153].classification[0] := 'M';
   additionalAlarmData[153].classification[1] := 'F';
   additionalAlarmData[153].classification[2..3] := ' ';
   additionalAlarmData[154].classification[0] := 'P';
   additionalAlarmData[154].classification[1] := 'F';
   additionalAlarmData[154].classification[2..3] := ' ';
   additionalAlarmData[155].classification[0] := 'T';
   additionalAlarmData[155].classification[1] := 'F';
   additionalAlarmData[155].classification[2] := 'I';
   additionalAlarmData[155].classification[3] := 'B';
   additionalAlarmData[156].classification[0] := 'T';
   additionalAlarmData[156].classification[1] := 'F';
   additionalAlarmData[156].classification[2] := 'S';
   additionalAlarmData[156].classification[3] := ' ';
   additionalAlarmData[157].classification[0] := 'S';
   additionalAlarmData[157].classification[1] := 'F';
   additionalAlarmData[157].classification[2..3] := ' ';
   additionalAlarmData[158].classification[0] := 'M';
   additionalAlarmData[158].classification[1] := 'W';
   additionalAlarmData[158].classification[2..3] := ' ';
   additionalAlarmData[159].classification[0] := 'P';
   additionalAlarmData[159].classification[1] := 'W';
   additionalAlarmData[159].classification[2..3] := ' ';
   additionalAlarmData[160].classification[0] := 'M';
   additionalAlarmData[160].classification[1] := 'S';
   additionalAlarmData[160].classification[2..3] := ' ';
   additionalAlarmData[161].classification[0] := 'M';
   additionalAlarmData[161].classification[1] := 'F';
   additionalAlarmData[161].classification[2..3] := ' ';
   additionalAlarmData[162].classification[0] := 'P';
   additionalAlarmData[162].classification[1] := 'F';
   additionalAlarmData[162].classification[2..3] := ' ';
   additionalAlarmData[163].classification[0] := 'T';
   additionalAlarmData[163].classification[1] := 'F';
   additionalAlarmData[163].classification[2] := 'I';
   additionalAlarmData[163].classification[3] := 'B';
   additionalAlarmData[164].classification[0] := 'T';
   additionalAlarmData[164].classification[1] := 'F';
   additionalAlarmData[164].classification[2] := 'S';
   additionalAlarmData[164].classification[3] := ' ';
   additionalAlarmData[165].classification[0] := 'S';
   additionalAlarmData[165].classification[1] := 'F';
   additionalAlarmData[165].classification[2..3] := ' ';
   additionalAlarmData[166].classification[0] := 'M';
   additionalAlarmData[166].classification[1] := 'W';
   additionalAlarmData[166].classification[2..3] := ' ';
   additionalAlarmData[167].classification[0] := 'P';
   additionalAlarmData[167].classification[1] := 'W';
   additionalAlarmData[167].classification[2..3] := ' ';
   additionalAlarmData[168].classification[0] := 'M';
   additionalAlarmData[168].classification[1] := 'S';
   additionalAlarmData[168].classification[2..3] := ' ';
   additionalAlarmData[169].classification[0] := 'S';
   additionalAlarmData[169].classification[1] := 'F';
   additionalAlarmData[169].classification[2..3] := ' ';
   additionalAlarmData[170].classification[0] := 'P';
   additionalAlarmData[170].classification[1] := 'F';
   additionalAlarmData[170].classification[2..3] := ' ';
   additionalAlarmData[171].classification[0] := 'T';
   additionalAlarmData[171].classification[1] := 'F';
   additionalAlarmData[171].classification[2] := 'I';
   additionalAlarmData[171].classification[3] := 'B';
   additionalAlarmData[172].classification[0] := 'T';
   additionalAlarmData[172].classification[1] := 'F';
   additionalAlarmData[172].classification[2] := 'S';
   additionalAlarmData[172].classification[3] := ' ';
   additionalAlarmData[173].classification[0] := 'S';
   additionalAlarmData[173].classification[1] := 'F';
   additionalAlarmData[173].classification[2..3] := ' ';
   additionalAlarmData[174].classification[0] := 'M';
   additionalAlarmData[174].classification[1] := 'W';
   additionalAlarmData[174].classification[2..3] := ' ';
   additionalAlarmData[175].classification[0] := 'P';
   additionalAlarmData[175].classification[1] := 'W';
   additionalAlarmData[175].classification[2..3] := ' ';
   additionalAlarmData[176].classification[0] := 'M';
   additionalAlarmData[176].classification[1] := 'S';
   additionalAlarmData[176].classification[2..3] := ' ';
   additionalAlarmData[177].classification[0..3] := ' ';
   additionalAlarmData[178].classification[0..3] := ' ';
   additionalAlarmData[179].classification[0..3] := ' ';
   additionalAlarmData[180].classification[0..3] := ' ';
   additionalAlarmData[181].classification[0..3] := ' ';
   additionalAlarmData[182].classification[0..3] := ' ';
   additionalAlarmData[183].classification[0..3] := ' ';
   additionalAlarmData[184].classification[0..3] := ' ';
   additionalAlarmData[185].classification[0..3] := ' ';
   additionalAlarmData[186].classification[0..3] := ' ';
   additionalAlarmData[187].classification[0..3] := ' ';
   additionalAlarmData[188].classification[0..3] := ' ';
   additionalAlarmData[189].classification[0..3] := ' ';
   additionalAlarmData[190].classification[0..3] := ' ';
   additionalAlarmData[191].classification[0..3] := ' ';
   additionalAlarmData[192].classification[0..3] := ' ';
   additionalAlarmData[193].classification[0..3] := ' ';
   additionalAlarmData[194].classification[0..3] := ' ';
   additionalAlarmData[195].classification[0..3] := ' ';
   additionalAlarmData[196].classification[0..3] := ' ';
   additionalAlarmData[197].classification[0..3] := ' ';
   additionalAlarmData[198].classification[0..3] := ' ';
   additionalAlarmData[199].classification[0..3] := ' ';
   additionalAlarmData[200].classification[0..3] := ' ';
   additionalAlarmData[201].classification[0..3] := ' ';
   additionalAlarmData[202].classification[0..3] := ' ';
   additionalAlarmData[203].classification[0..3] := ' ';
   additionalAlarmData[204].classification[0..3] := ' ';
   additionalAlarmData[205].classification[0..3] := ' ';
   additionalAlarmData[206].classification[0..3] := ' ';
   additionalAlarmData[207].classification[0..3] := ' ';
   additionalAlarmData[208].classification[0..3] := ' ';
   additionalAlarmData[209].classification[0..3] := ' ';
   additionalAlarmData[210].classification[0..3] := ' ';
   additionalAlarmData[211].classification[0..3] := ' ';
   additionalAlarmData[212].classification[0..3] := ' ';
   additionalAlarmData[213].classification[0..3] := ' ';
   additionalAlarmData[214].classification[0..3] := ' ';
   additionalAlarmData[215].classification[0..3] := ' ';
   additionalAlarmData[216].classification[0..3] := ' ';
   additionalAlarmData[217].classification[0..3] := ' ';
   additionalAlarmData[218].classification[0..3] := ' ';
   additionalAlarmData[219].classification[0..3] := ' ';
   additionalAlarmData[220].classification[0..3] := ' ';
   additionalAlarmData[221].classification[0..3] := ' ';
   additionalAlarmData[222].classification[0..3] := ' ';
   additionalAlarmData[223].classification[0..3] := ' ';
   additionalAlarmData[224].classification[0..3] := ' ';
   additionalAlarmData[225].classification[0..3] := ' ';
   additionalAlarmData[226].classification[0..3] := ' ';
   additionalAlarmData[227].classification[0..3] := ' ';
   additionalAlarmData[228].classification[0..3] := ' ';
   additionalAlarmData[229].classification[0..3] := ' ';
   additionalAlarmData[230].classification[0..3] := ' ';
   additionalAlarmData[231].classification[0..3] := ' ';
   additionalAlarmData[232].classification[0..3] := ' ';
   additionalAlarmData[233].classification[0..3] := ' ';
   additionalAlarmData[234].classification[0..3] := ' ';
   additionalAlarmData[235].classification[0..3] := ' ';
   additionalAlarmData[236].classification[0..3] := ' ';
   additionalAlarmData[237].classification[0..3] := ' ';
   additionalAlarmData[238].classification[0..3] := ' ';
   additionalAlarmData[239].classification[0..3] := ' ';
   additionalAlarmData[240].classification[0..3] := ' ';
   additionalAlarmData[241].classification[0..3] := ' ';
   additionalAlarmData[242].classification[0..3] := ' ';
   additionalAlarmData[243].classification[0..3] := ' ';
   additionalAlarmData[244].classification[0..3] := ' ';
   additionalAlarmData[245].classification[0..3] := ' ';
   additionalAlarmData[246].classification[0..3] := ' ';
   additionalAlarmData[247].classification[0..3] := ' ';
   additionalAlarmData[248].classification[0..3] := ' ';
   additionalAlarmData[249].classification[0..3] := ' ';
   additionalAlarmData[250].classification[0..3] := ' ';
   additionalAlarmData[251].classification[0..3] := ' ';
   additionalAlarmData[252].classification[0..3] := ' ';
   additionalAlarmData[253].classification[0..3] := ' ';
   additionalAlarmData[254].classification[0..3] := ' ';
   additionalAlarmData[255].classification[0..3] := ' ';
   additionalAlarmData[256].classification[0..3] := ' ';
   additionalAlarmData[257].classification[0..3] := ' ';
   additionalAlarmData[258].classification[0..3] := ' ';
   additionalAlarmData[259].classification[0..3] := ' ';
   additionalAlarmData[260].classification[0..3] := ' ';
   additionalAlarmData[261].classification[0..3] := ' ';
   additionalAlarmData[262].classification[0..3] := ' ';
   additionalAlarmData[263].classification[0..3] := ' ';
   additionalAlarmData[264].classification[0..3] := ' ';
   additionalAlarmData[265].classification[0..3] := ' ';
   additionalAlarmData[266].classification[0..3] := ' ';
   additionalAlarmData[267].classification[0..3] := ' ';
   additionalAlarmData[268].classification[0..3] := ' ';
   additionalAlarmData[269].classification[0..3] := ' ';
   additionalAlarmData[270].classification[0..3] := ' ';
   additionalAlarmData[271].classification[0..3] := ' ';
   additionalAlarmData[272].classification[0..3] := ' ';
   additionalAlarmData[273].classification[0..3] := ' ';
   additionalAlarmData[274].classification[0..3] := ' ';
   additionalAlarmData[275].classification[0..3] := ' ';
   additionalAlarmData[276].classification[0..3] := ' ';
   additionalAlarmData[277].classification[0..3] := ' ';
   additionalAlarmData[278].classification[0..3] := ' ';
   additionalAlarmData[279].classification[0..3] := ' ';
   additionalAlarmData[280].classification[0..3] := ' ';
   additionalAlarmData[281].classification[0..3] := ' ';
   additionalAlarmData[282].classification[0..3] := ' ';
   additionalAlarmData[283].classification[0..3] := ' ';
   additionalAlarmData[284].classification[0..3] := ' ';
   additionalAlarmData[285].classification[0..3] := ' ';
   additionalAlarmData[286].classification[0..3] := ' ';
   additionalAlarmData[287].classification[0..3] := ' ';
   additionalAlarmData[288].classification[0..3] := ' ';
   additionalAlarmData[289].classification[0..3] := ' ';
   additionalAlarmData[290].classification[0..3] := ' ';
   additionalAlarmData[291].classification[0..3] := ' ';
   additionalAlarmData[292].classification[0..3] := ' ';
   additionalAlarmData[293].classification[0..3] := ' ';
   additionalAlarmData[294].classification[0..3] := ' ';
   additionalAlarmData[295].classification[0..3] := ' ';
   additionalAlarmData[296].classification[0..3] := ' ';
   additionalAlarmData[297].classification[0..3] := ' ';
   additionalAlarmData[298].classification[0..3] := ' ';
   additionalAlarmData[299].classification[0..3] := ' ';
   additionalAlarmData[300].classification[0..3] := ' ';
   additionalAlarmData[301].classification[0..3] := ' ';
   additionalAlarmData[302].classification[0..3] := ' ';
   additionalAlarmData[303].classification[0..3] := ' ';
   additionalAlarmData[304].classification[0..3] := ' ';
   additionalAlarmData[305].classification[0..3] := ' ';
   additionalAlarmData[306].classification[0..3] := ' ';
   additionalAlarmData[307].classification[0..3] := ' ';
   additionalAlarmData[308].classification[0..3] := ' ';
   additionalAlarmData[309].classification[0..3] := ' ';
   additionalAlarmData[310].classification[0..3] := ' ';
   additionalAlarmData[311].classification[0..3] := ' ';
   additionalAlarmData[312].classification[0..3] := ' ';
   additionalAlarmData[313].classification[0..3] := ' ';
   additionalAlarmData[314].classification[0..3] := ' ';
   additionalAlarmData[315].classification[0..3] := ' ';
   additionalAlarmData[316].classification[0..3] := ' ';
   additionalAlarmData[317].classification[0..3] := ' ';
   additionalAlarmData[318].classification[0..3] := ' ';
   additionalAlarmData[319].classification[0..3] := ' ';
   additionalAlarmData[320].classification[0..3] := ' ';
   additionalAlarmData[321].classification[0..3] := ' ';
   additionalAlarmData[322].classification[0..3] := ' ';
   additionalAlarmData[323].classification[0..3] := ' ';
   additionalAlarmData[324].classification[0..3] := ' ';
   additionalAlarmData[325].classification[0..3] := ' ';
   additionalAlarmData[326].classification[0..3] := ' ';
   additionalAlarmData[327].classification[0..3] := ' ';
   additionalAlarmData[328].classification[0..3] := ' ';
   additionalAlarmData[329].classification[0..3] := ' ';
   additionalAlarmData[330].classification[0..3] := ' ';
   additionalAlarmData[331].classification[0..3] := ' ';
   additionalAlarmData[332].classification[0..3] := ' ';
   additionalAlarmData[333].classification[0..3] := ' ';
   additionalAlarmData[334].classification[0..3] := ' ';
   additionalAlarmData[335].classification[0..3] := ' ';
   additionalAlarmData[336].classification[0..3] := ' ';
   additionalAlarmData[337].classification[0..3] := ' ';
   additionalAlarmData[338].classification[0..3] := ' ';
   additionalAlarmData[339].classification[0..3] := ' ';
   additionalAlarmData[340].classification[0..3] := ' ';
   additionalAlarmData[341].classification[0..3] := ' ';
   additionalAlarmData[342].classification[0..3] := ' ';
   additionalAlarmData[343].classification[0..3] := ' ';
   additionalAlarmData[344].classification[0..3] := ' ';
   additionalAlarmData[345].classification[0..3] := ' ';
   additionalAlarmData[346].classification[0..3] := ' ';
   additionalAlarmData[347].classification[0..3] := ' ';
   additionalAlarmData[348].classification[0..3] := ' ';
   additionalAlarmData[349].classification[0..3] := ' ';
   additionalAlarmData[350].classification[0..3] := ' ';
   additionalAlarmData[351].classification[0..3] := ' ';
   additionalAlarmData[352].classification[0..3] := ' ';
   additionalAlarmData[353].classification[0..3] := ' ';
   additionalAlarmData[354].classification[0..3] := ' ';
   additionalAlarmData[355].classification[0..3] := ' ';
   additionalAlarmData[356].classification[0..3] := ' ';
   additionalAlarmData[357].classification[0..3] := ' ';
   additionalAlarmData[358].classification[0..3] := ' ';
   additionalAlarmData[359].classification[0..3] := ' ';
   additionalAlarmData[360].classification[0..3] := ' ';
   additionalAlarmData[361].classification[0..3] := ' ';
   additionalAlarmData[362].classification[0..3] := ' ';
   additionalAlarmData[363].classification[0..3] := ' ';
   additionalAlarmData[364].classification[0..3] := ' ';
   additionalAlarmData[365].classification[0..3] := ' ';
   additionalAlarmData[366].classification[0..3] := ' ';
   additionalAlarmData[367].classification[0..3] := ' ';
   additionalAlarmData[368].classification[0..3] := ' ';
   additionalAlarmData[369].classification[0..3] := ' ';
   additionalAlarmData[370].classification[0..3] := ' ';
   additionalAlarmData[371].classification[0..3] := ' ';
   additionalAlarmData[372].classification[0..3] := ' ';
   additionalAlarmData[373].classification[0..3] := ' ';
   additionalAlarmData[374].classification[0..3] := ' ';
   additionalAlarmData[375].classification[0..3] := ' ';
   additionalAlarmData[376].classification[0..3] := ' ';
   additionalAlarmData[377].classification[0..3] := ' ';
   additionalAlarmData[378].classification[0..3] := ' ';
   additionalAlarmData[379].classification[0..3] := ' ';
   additionalAlarmData[380].classification[0..3] := ' ';
   additionalAlarmData[381].classification[0..3] := ' ';
   additionalAlarmData[382].classification[0..3] := ' ';
   additionalAlarmData[383].classification[0..3] := ' ';
   additionalAlarmData[384].classification[0..3] := ' ';
   additionalAlarmData[385].classification[0..3] := ' ';
   additionalAlarmData[386].classification[0..3] := ' ';
   additionalAlarmData[387].classification[0..3] := ' ';
   additionalAlarmData[388].classification[0..3] := ' ';
   additionalAlarmData[389].classification[0..3] := ' ';
   additionalAlarmData[390].classification[0..3] := ' ';
   additionalAlarmData[391].classification[0..3] := ' ';
   additionalAlarmData[392].classification[0..3] := ' ';
   additionalAlarmData[393].classification[0..3] := ' ';
   additionalAlarmData[394].classification[0..3] := ' ';
   additionalAlarmData[395].classification[0..3] := ' ';
   additionalAlarmData[396].classification[0..3] := ' ';
   additionalAlarmData[397].classification[0..3] := ' ';
   additionalAlarmData[398].classification[0..3] := ' ';
   additionalAlarmData[399].classification[0..3] := ' ';
   additionalAlarmData[400].classification[0..3] := ' ';
   additionalAlarmData[401].classification[0..3] := ' ';
   additionalAlarmData[402].classification[0..3] := ' ';
   additionalAlarmData[403].classification[0..3] := ' ';
   additionalAlarmData[404].classification[0..3] := ' ';
   additionalAlarmData[405].classification[0..3] := ' ';
   additionalAlarmData[406].classification[0..3] := ' ';
   additionalAlarmData[407].classification[0..3] := ' ';
   additionalAlarmData[408].classification[0..3] := ' ';
   additionalAlarmData[409].classification[0..3] := ' ';
   additionalAlarmData[410].classification[0..3] := ' ';
   additionalAlarmData[411].classification[0..3] := ' ';
   additionalAlarmData[412].classification[0..3] := ' ';
   additionalAlarmData[413].classification[0..3] := ' ';
   additionalAlarmData[414].classification[0..3] := ' ';
   additionalAlarmData[415].classification[0..3] := ' ';
   additionalAlarmData[416].classification[0..3] := ' ';
   additionalAlarmData[417].classification[0..3] := ' ';
   additionalAlarmData[418].classification[0..3] := ' ';
   additionalAlarmData[419].classification[0..3] := ' ';
   additionalAlarmData[420].classification[0..3] := ' ';
   additionalAlarmData[421].classification[0..3] := ' ';
   additionalAlarmData[422].classification[0..3] := ' ';
   additionalAlarmData[423].classification[0..3] := ' ';
   additionalAlarmData[424].classification[0..3] := ' ';
   additionalAlarmData[425].classification[0..3] := ' ';
   additionalAlarmData[426].classification[0..3] := ' ';
   additionalAlarmData[427].classification[0..3] := ' ';
   additionalAlarmData[428].classification[0..3] := ' ';
   additionalAlarmData[429].classification[0..3] := ' ';
   additionalAlarmData[430].classification[0..3] := ' ';
   additionalAlarmData[431].classification[0..3] := ' ';
   additionalAlarmData[432].classification[0..3] := ' ';
   additionalAlarmData[433].classification[0..3] := ' ';
   additionalAlarmData[434].classification[0..3] := ' ';
   additionalAlarmData[435].classification[0..3] := ' ';
   additionalAlarmData[436].classification[0..3] := ' ';
   additionalAlarmData[437].classification[0..3] := ' ';
   additionalAlarmData[438].classification[0..3] := ' ';
   additionalAlarmData[439].classification[0..3] := ' ';
   additionalAlarmData[440].classification[0..3] := ' ';
   additionalAlarmData[441].classification[0..3] := ' ';
   additionalAlarmData[442].classification[0..3] := ' ';
   additionalAlarmData[443].classification[0..3] := ' ';
   additionalAlarmData[444].classification[0..3] := ' ';
   additionalAlarmData[445].classification[0..3] := ' ';
   additionalAlarmData[446].classification[0..3] := ' ';
   additionalAlarmData[447].classification[0..3] := ' ';
   additionalAlarmData[448].classification[0..3] := ' ';
   additionalAlarmData[449].classification[0..3] := ' ';
   additionalAlarmData[450].classification[0..3] := ' ';
   additionalAlarmData[451].classification[0..3] := ' ';
   additionalAlarmData[452].classification[0..3] := ' ';
   additionalAlarmData[453].classification[0..3] := ' ';
   additionalAlarmData[454].classification[0..3] := ' ';
   additionalAlarmData[455].classification[0..3] := ' ';
   additionalAlarmData[456].classification[0..3] := ' ';
   additionalAlarmData[457].classification[0..3] := ' ';
   additionalAlarmData[458].classification[0..3] := ' ';
   additionalAlarmData[459].classification[0..3] := ' ';
   additionalAlarmData[460].classification[0..3] := ' ';
   additionalAlarmData[461].classification[0..3] := ' ';
   additionalAlarmData[462].classification[0..3] := ' ';
   additionalAlarmData[463].classification[0..3] := ' ';
   additionalAlarmData[464].classification[0..3] := ' ';
   additionalAlarmData[465].classification[0..3] := ' ';
   additionalAlarmData[466].classification[0..3] := ' ';
   additionalAlarmData[467].classification[0..3] := ' ';
   additionalAlarmData[468].classification[0..3] := ' ';
   additionalAlarmData[469].classification[0..3] := ' ';
   additionalAlarmData[470].classification[0..3] := ' ';
   additionalAlarmData[471].classification[0..3] := ' ';
   additionalAlarmData[472].classification[0..3] := ' ';
   additionalAlarmData[473].classification[0..3] := ' ';
   additionalAlarmData[474].classification[0..3] := ' ';
   additionalAlarmData[475].classification[0..3] := ' ';
   additionalAlarmData[476].classification[0..3] := ' ';
   additionalAlarmData[477].classification[0..3] := ' ';
   additionalAlarmData[478].classification[0..3] := ' ';
   additionalAlarmData[479].classification[0..3] := ' ';
   additionalAlarmData[480].classification[0..3] := ' ';
   additionalAlarmData[481].classification[0..3] := ' ';
   additionalAlarmData[482].classification[0..3] := ' ';
   additionalAlarmData[483].classification[0..3] := ' ';
   additionalAlarmData[484].classification[0..3] := ' ';
   additionalAlarmData[485].classification[0..3] := ' ';
   additionalAlarmData[486].classification[0..3] := ' ';
   additionalAlarmData[487].classification[0..3] := ' ';
   additionalAlarmData[488].classification[0..3] := ' ';
   additionalAlarmData[489].classification[0..3] := ' ';
   additionalAlarmData[490].classification[0..3] := ' ';
   additionalAlarmData[491].classification[0..3] := ' ';
   additionalAlarmData[492].classification[0..3] := ' ';
   additionalAlarmData[493].classification[0..3] := ' ';
   additionalAlarmData[494].classification[0..3] := ' ';
   additionalAlarmData[495].classification[0..3] := ' ';
   additionalAlarmData[496].classification[0..3] := ' ';
   additionalAlarmData[497].classification[0..3] := ' ';
   additionalAlarmData[498].classification[0..3] := ' ';
   additionalAlarmData[499].classification[0..3] := ' ';
   additionalAlarmData[500].classification[0] := 'M';
   additionalAlarmData[500].classification[1] := 'F';
   additionalAlarmData[500].classification[2..3] := ' ';
   additionalAlarmData[501].classification[0..3] := ' ';
   additionalAlarmData[502].classification[0..3] := ' ';
   additionalAlarmData[503].classification[0..3] := ' ';
   additionalAlarmData[504].classification[0..3] := ' ';
   additionalAlarmData[505].classification[0..3] := ' ';
   additionalAlarmData[506].classification[0..3] := ' ';
   additionalAlarmData[507].classification[0..3] := ' ';
   additionalAlarmData[508].classification[0..3] := ' ';
   additionalAlarmData[509].classification[0..3] := ' ';
   additionalAlarmData[510].classification[0..3] := ' ';
   additionalAlarmData[511].classification[0..3] := ' ';
   additionalAlarmData[512].classification[0..3] := ' ';
   additionalAlarmData[513].classification[0..3] := ' ';
   additionalAlarmData[514].classification[0..3] := ' ';
   additionalAlarmData[515].classification[0..3] := ' ';
   additionalAlarmData[516].classification[0..3] := ' ';
   additionalAlarmData[517].classification[0..3] := ' ';
   additionalAlarmData[518].classification[0..3] := ' ';
   additionalAlarmData[519].classification[0..3] := ' ';
   additionalAlarmData[520].classification[0..3] := ' ';
   additionalAlarmData[521].classification[0..3] := ' ';
   additionalAlarmData[522].classification[0..3] := ' ';
   additionalAlarmData[523].classification[0..3] := ' ';
   additionalAlarmData[524].classification[0..3] := ' ';
   additionalAlarmData[525].classification[0..3] := ' ';
   additionalAlarmData[526].classification[0..3] := ' ';
   additionalAlarmData[527].classification[0..3] := ' ';
   additionalAlarmData[528].classification[0..3] := ' ';
   additionalAlarmData[529].classification[0..3] := ' ';
   additionalAlarmData[530].classification[0..3] := ' ';
   additionalAlarmData[531].classification[0..3] := ' ';
   additionalAlarmData[532].classification[0..3] := ' ';
   additionalAlarmData[533].classification[0..3] := ' ';
   additionalAlarmData[534].classification[0..3] := ' ';
   additionalAlarmData[535].classification[0..3] := ' ';
   additionalAlarmData[536].classification[0..3] := ' ';
   additionalAlarmData[537].classification[0..3] := ' ';
   additionalAlarmData[538].classification[0..3] := ' ';
   additionalAlarmData[539].classification[0..3] := ' ';
   additionalAlarmData[540].classification[0..3] := ' ';
   additionalAlarmData[541].classification[0..3] := ' ';
   additionalAlarmData[542].classification[0..3] := ' ';
   additionalAlarmData[543].classification[0..3] := ' ';
   additionalAlarmData[544].classification[0..3] := ' ';
   additionalAlarmData[545].classification[0..3] := ' ';
   additionalAlarmData[546].classification[0..3] := ' ';
   additionalAlarmData[547].classification[0..3] := ' ';
   additionalAlarmData[548].classification[0..3] := ' ';
   additionalAlarmData[549].classification[0..3] := ' ';
   additionalAlarmData[550].classification[0..3] := ' ';
   additionalAlarmData[551].classification[0..3] := ' ';
   additionalAlarmData[552].classification[0..3] := ' ';
   additionalAlarmData[553].classification[0..3] := ' ';
   additionalAlarmData[554].classification[0..3] := ' ';
   additionalAlarmData[555].classification[0..3] := ' ';
   additionalAlarmData[556].classification[0..3] := ' ';
   additionalAlarmData[557].classification[0..3] := ' ';
   additionalAlarmData[558].classification[0..3] := ' ';
   additionalAlarmData[559].classification[0..3] := ' ';
   additionalAlarmData[560].classification[0..3] := ' ';
   additionalAlarmData[561].classification[0..3] := ' ';
   additionalAlarmData[562].classification[0..3] := ' ';
   additionalAlarmData[563].classification[0..3] := ' ';
   additionalAlarmData[564].classification[0..3] := ' ';
   additionalAlarmData[565].classification[0..3] := ' ';
   additionalAlarmData[566].classification[0..3] := ' ';
   additionalAlarmData[567].classification[0..3] := ' ';
   additionalAlarmData[568].classification[0..3] := ' ';
   additionalAlarmData[569].classification[0..3] := ' ';
   additionalAlarmData[570].classification[0..3] := ' ';
   additionalAlarmData[571].classification[0..3] := ' ';
   additionalAlarmData[572].classification[0..3] := ' ';
   additionalAlarmData[573].classification[0..3] := ' ';
   additionalAlarmData[574].classification[0..3] := ' ';
   additionalAlarmData[575].classification[0..3] := ' ';
   additionalAlarmData[576].classification[0..3] := ' ';
   additionalAlarmData[577].classification[0..3] := ' ';
   additionalAlarmData[578].classification[0..3] := ' ';
   additionalAlarmData[579].classification[0..3] := ' ';
   additionalAlarmData[580].classification[0..3] := ' ';
   additionalAlarmData[581].classification[0..3] := ' ';
   additionalAlarmData[582].classification[0..3] := ' ';
   additionalAlarmData[583].classification[0..3] := ' ';
   additionalAlarmData[584].classification[0..3] := ' ';
   additionalAlarmData[585].classification[0..3] := ' ';
   additionalAlarmData[586].classification[0..3] := ' ';
   additionalAlarmData[587].classification[0..3] := ' ';
   additionalAlarmData[588].classification[0..3] := ' ';
   additionalAlarmData[589].classification[0..3] := ' ';
   additionalAlarmData[590].classification[0..3] := ' ';
   additionalAlarmData[591].classification[0..3] := ' ';
   additionalAlarmData[592].classification[0..3] := ' ';
   additionalAlarmData[593].classification[0..3] := ' ';
   additionalAlarmData[594].classification[0..3] := ' ';
   additionalAlarmData[595].classification[0..3] := ' ';
   additionalAlarmData[596].classification[0..3] := ' ';
   additionalAlarmData[597].classification[0..3] := ' ';
   additionalAlarmData[598].classification[0..3] := ' ';
   additionalAlarmData[599].classification[0..3] := ' ';
   additionalAlarmData[600].classification[0..3] := ' ';
   additionalAlarmData[601].classification[0..3] := ' ';
   additionalAlarmData[602].classification[0..3] := ' ';
   additionalAlarmData[603].classification[0..3] := ' ';
   additionalAlarmData[604].classification[0..3] := ' ';
   additionalAlarmData[605].classification[0..3] := ' ';
   additionalAlarmData[606].classification[0..3] := ' ';
   additionalAlarmData[607].classification[0..3] := ' ';
   additionalAlarmData[608].classification[0..3] := ' ';
   additionalAlarmData[609].classification[0..3] := ' ';
   additionalAlarmData[610].classification[0..3] := ' ';
   additionalAlarmData[611].classification[0..3] := ' ';
   additionalAlarmData[612].classification[0..3] := ' ';
   additionalAlarmData[613].classification[0..3] := ' ';
   additionalAlarmData[614].classification[0..3] := ' ';
   additionalAlarmData[615].classification[0..3] := ' ';
   additionalAlarmData[616].classification[0..3] := ' ';
   additionalAlarmData[617].classification[0..3] := ' ';
   additionalAlarmData[618].classification[0..3] := ' ';
   additionalAlarmData[619].classification[0..3] := ' ';
   additionalAlarmData[620].classification[0..3] := ' ';
   additionalAlarmData[621].classification[0..3] := ' ';
   additionalAlarmData[622].classification[0..3] := ' ';
   additionalAlarmData[623].classification[0..3] := ' ';
   additionalAlarmData[624].classification[0..3] := ' ';
   additionalAlarmData[625].classification[0..3] := ' ';
   additionalAlarmData[626].classification[0..3] := ' ';
   additionalAlarmData[627].classification[0..3] := ' ';
   additionalAlarmData[628].classification[0..3] := ' ';
   additionalAlarmData[629].classification[0..3] := ' ';
   additionalAlarmData[630].classification[0..3] := ' ';
   additionalAlarmData[631].classification[0..3] := ' ';
   additionalAlarmData[632].classification[0..3] := ' ';
   additionalAlarmData[633].classification[0..3] := ' ';
   additionalAlarmData[634].classification[0..3] := ' ';
   additionalAlarmData[635].classification[0..3] := ' ';
   additionalAlarmData[636].classification[0..3] := ' ';
   additionalAlarmData[637].classification[0..3] := ' ';
   additionalAlarmData[638].classification[0..3] := ' ';
   additionalAlarmData[639].classification[0..3] := ' ';
   additionalAlarmData[640].classification[0..3] := ' ';
   additionalAlarmData[641].classification[0..3] := ' ';
   additionalAlarmData[642].classification[0..3] := ' ';
   additionalAlarmData[643].classification[0..3] := ' ';
   additionalAlarmData[644].classification[0..3] := ' ';
   additionalAlarmData[645].classification[0..3] := ' ';
   additionalAlarmData[646].classification[0..3] := ' ';
   additionalAlarmData[647].classification[0..3] := ' ';
   additionalAlarmData[648].classification[0..3] := ' ';
   additionalAlarmData[649].classification[0..3] := ' ';
   additionalAlarmData[650].classification[0..3] := ' ';
   additionalAlarmData[651].classification[0..3] := ' ';
   additionalAlarmData[652].classification[0..3] := ' ';
   additionalAlarmData[653].classification[0..3] := ' ';
   additionalAlarmData[654].classification[0..3] := ' ';
   additionalAlarmData[655].classification[0..3] := ' ';
   additionalAlarmData[656].classification[0..3] := ' ';
   additionalAlarmData[657].classification[0..3] := ' ';
   additionalAlarmData[658].classification[0..3] := ' ';
   additionalAlarmData[659].classification[0..3] := ' ';
   additionalAlarmData[660].classification[0..3] := ' ';
   additionalAlarmData[661].classification[0..3] := ' ';
   additionalAlarmData[662].classification[0..3] := ' ';
   additionalAlarmData[663].classification[0..3] := ' ';
   additionalAlarmData[664].classification[0..3] := ' ';
   additionalAlarmData[665].classification[0..3] := ' ';
   additionalAlarmData[666].classification[0..3] := ' ';
   additionalAlarmData[667].classification[0..3] := ' ';
   additionalAlarmData[668].classification[0..3] := ' ';
   additionalAlarmData[669].classification[0..3] := ' ';
   additionalAlarmData[670].classification[0..3] := ' ';
   additionalAlarmData[671].classification[0..3] := ' ';
   additionalAlarmData[672].classification[0..3] := ' ';
   additionalAlarmData[673].classification[0..3] := ' ';
   additionalAlarmData[674].classification[0..3] := ' ';
   additionalAlarmData[675].classification[0..3] := ' ';
   additionalAlarmData[676].classification[0..3] := ' ';
   additionalAlarmData[677].classification[0..3] := ' ';
   additionalAlarmData[678].classification[0..3] := ' ';
   additionalAlarmData[679].classification[0..3] := ' ';
   additionalAlarmData[680].classification[0..3] := ' ';
   additionalAlarmData[681].classification[0..3] := ' ';
   additionalAlarmData[682].classification[0..3] := ' ';
   additionalAlarmData[683].classification[0..3] := ' ';
   additionalAlarmData[684].classification[0..3] := ' ';
   additionalAlarmData[685].classification[0..3] := ' ';
   additionalAlarmData[686].classification[0..3] := ' ';
   additionalAlarmData[687].classification[0..3] := ' ';
   additionalAlarmData[688].classification[0..3] := ' ';
   additionalAlarmData[689].classification[0..3] := ' ';
   additionalAlarmData[690].classification[0..3] := ' ';
   additionalAlarmData[691].classification[0..3] := ' ';
   additionalAlarmData[692].classification[0..3] := ' ';
   additionalAlarmData[693].classification[0..3] := ' ';
   additionalAlarmData[694].classification[0..3] := ' ';
   additionalAlarmData[695].classification[0..3] := ' ';
   additionalAlarmData[696].classification[0..3] := ' ';
   additionalAlarmData[697].classification[0..3] := ' ';
   additionalAlarmData[698].classification[0..3] := ' ';
   additionalAlarmData[699].classification[0..3] := ' ';
   additionalAlarmData[700].classification[0..3] := ' ';
   additionalAlarmData[701].classification[0..3] := ' ';
   additionalAlarmData[702].classification[0..3] := ' ';
   additionalAlarmData[703].classification[0..3] := ' ';
   additionalAlarmData[704].classification[0..3] := ' ';
   additionalAlarmData[705].classification[0..3] := ' ';
   additionalAlarmData[706].classification[0..3] := ' ';
   additionalAlarmData[707].classification[0..3] := ' ';
   additionalAlarmData[708].classification[0..3] := ' ';
   additionalAlarmData[709].classification[0..3] := ' ';
   additionalAlarmData[710].classification[0..3] := ' ';
   additionalAlarmData[711].classification[0..3] := ' ';
   additionalAlarmData[712].classification[0..3] := ' ';
   additionalAlarmData[713].classification[0..3] := ' ';
   additionalAlarmData[714].classification[0..3] := ' ';
   additionalAlarmData[715].classification[0..3] := ' ';
   additionalAlarmData[716].classification[0..3] := ' ';
   additionalAlarmData[717].classification[0..3] := ' ';
   additionalAlarmData[718].classification[0..3] := ' ';
   additionalAlarmData[719].classification[0..3] := ' ';
   additionalAlarmData[720].classification[0..3] := ' ';
   additionalAlarmData[721].classification[0..3] := ' ';
   additionalAlarmData[722].classification[0..3] := ' ';
   additionalAlarmData[723].classification[0..3] := ' ';
   additionalAlarmData[724].classification[0..3] := ' ';
   additionalAlarmData[725].classification[0..3] := ' ';
   additionalAlarmData[726].classification[0..3] := ' ';
   additionalAlarmData[727].classification[0..3] := ' ';
   additionalAlarmData[728].classification[0..3] := ' ';
   additionalAlarmData[729].classification[0..3] := ' ';
   additionalAlarmData[730].classification[0..3] := ' ';
   additionalAlarmData[731].classification[0..3] := ' ';
   additionalAlarmData[732].classification[0..3] := ' ';
   additionalAlarmData[733].classification[0..3] := ' ';
   additionalAlarmData[734].classification[0..3] := ' ';
   additionalAlarmData[735].classification[0..3] := ' ';
   additionalAlarmData[736].classification[0..3] := ' ';
   additionalAlarmData[737].classification[0..3] := ' ';
   additionalAlarmData[738].classification[0..3] := ' ';
   additionalAlarmData[739].classification[0..3] := ' ';
   additionalAlarmData[740].classification[0..3] := ' ';
   additionalAlarmData[741].classification[0..3] := ' ';
   additionalAlarmData[742].classification[0..3] := ' ';
   additionalAlarmData[743].classification[0..3] := ' ';
   additionalAlarmData[744].classification[0..3] := ' ';
   additionalAlarmData[745].classification[0..3] := ' ';
   additionalAlarmData[746].classification[0..3] := ' ';
   additionalAlarmData[747].classification[0..3] := ' ';
   additionalAlarmData[748].classification[0..3] := ' ';
   additionalAlarmData[749].classification[0..3] := ' ';
   additionalAlarmData[750].classification[0..3] := ' ';
   additionalAlarmData[751].classification[0..3] := ' ';
   additionalAlarmData[752].classification[0..3] := ' ';
   additionalAlarmData[753].classification[0..3] := ' ';
   additionalAlarmData[754].classification[0..3] := ' ';
   additionalAlarmData[755].classification[0..3] := ' ';
   additionalAlarmData[756].classification[0..3] := ' ';
   additionalAlarmData[757].classification[0..3] := ' ';
   additionalAlarmData[758].classification[0..3] := ' ';
   additionalAlarmData[759].classification[0..3] := ' ';
   additionalAlarmData[760].classification[0..3] := ' ';
   additionalAlarmData[761].classification[0..3] := ' ';
   additionalAlarmData[762].classification[0..3] := ' ';
   additionalAlarmData[763].classification[0..3] := ' ';
   additionalAlarmData[764].classification[0..3] := ' ';
   additionalAlarmData[765].classification[0..3] := ' ';
   additionalAlarmData[766].classification[0..3] := ' ';
   additionalAlarmData[767].classification[0..3] := ' ';
   additionalAlarmData[768].classification[0..3] := ' ';
   additionalAlarmData[769].classification[0..3] := ' ';
   additionalAlarmData[770].classification[0..3] := ' ';
   additionalAlarmData[771].classification[0..3] := ' ';
   additionalAlarmData[772].classification[0..3] := ' ';
   additionalAlarmData[773].classification[0..3] := ' ';
   additionalAlarmData[774].classification[0..3] := ' ';
   additionalAlarmData[775].classification[0..3] := ' ';
   additionalAlarmData[776].classification[0..3] := ' ';
   additionalAlarmData[777].classification[0..3] := ' ';
   additionalAlarmData[778].classification[0..3] := ' ';
   additionalAlarmData[779].classification[0..3] := ' ';
   additionalAlarmData[780].classification[0..3] := ' ';
   additionalAlarmData[781].classification[0..3] := ' ';
   additionalAlarmData[782].classification[0..3] := ' ';
   additionalAlarmData[783].classification[0..3] := ' ';
   additionalAlarmData[784].classification[0..3] := ' ';
   additionalAlarmData[785].classification[0..3] := ' ';
   additionalAlarmData[786].classification[0..3] := ' ';
   additionalAlarmData[787].classification[0..3] := ' ';
   additionalAlarmData[788].classification[0..3] := ' ';
   additionalAlarmData[789].classification[0..3] := ' ';
   additionalAlarmData[790].classification[0..3] := ' ';
   additionalAlarmData[791].classification[0..3] := ' ';
   additionalAlarmData[792].classification[0..3] := ' ';
   additionalAlarmData[793].classification[0..3] := ' ';
   additionalAlarmData[794].classification[0..3] := ' ';
   additionalAlarmData[795].classification[0..3] := ' ';
   additionalAlarmData[796].classification[0..3] := ' ';
   additionalAlarmData[797].classification[0..3] := ' ';
   additionalAlarmData[798].classification[0..3] := ' ';
   additionalAlarmData[799].classification[0..3] := ' ';
   additionalAlarmData[800].classification[0..3] := ' ';
   additionalAlarmData[801].classification[0..3] := ' ';
   additionalAlarmData[802].classification[0..3] := ' ';
   additionalAlarmData[803].classification[0..3] := ' ';
   additionalAlarmData[804].classification[0..3] := ' ';
   additionalAlarmData[805].classification[0..3] := ' ';
   additionalAlarmData[806].classification[0..3] := ' ';
   additionalAlarmData[807].classification[0..3] := ' ';
   additionalAlarmData[808].classification[0..3] := ' ';
   additionalAlarmData[809].classification[0..3] := ' ';
   additionalAlarmData[810].classification[0..3] := ' ';
   additionalAlarmData[811].classification[0..3] := ' ';
   additionalAlarmData[812].classification[0..3] := ' ';
   additionalAlarmData[813].classification[0..3] := ' ';
   additionalAlarmData[814].classification[0..3] := ' ';
   additionalAlarmData[815].classification[0..3] := ' ';
   additionalAlarmData[816].classification[0..3] := ' ';
   additionalAlarmData[817].classification[0..3] := ' ';
   additionalAlarmData[818].classification[0..3] := ' ';
   additionalAlarmData[819].classification[0..3] := ' ';
   additionalAlarmData[820].classification[0..3] := ' ';
   additionalAlarmData[821].classification[0..3] := ' ';
   additionalAlarmData[822].classification[0..3] := ' ';
   additionalAlarmData[823].classification[0..3] := ' ';
   additionalAlarmData[824].classification[0..3] := ' ';
   additionalAlarmData[825].classification[0..3] := ' ';
   additionalAlarmData[826].classification[0..3] := ' ';
   additionalAlarmData[827].classification[0..3] := ' ';
   additionalAlarmData[828].classification[0..3] := ' ';
   additionalAlarmData[829].classification[0..3] := ' ';
   additionalAlarmData[830].classification[0..3] := ' ';
   additionalAlarmData[831].classification[0..3] := ' ';
   additionalAlarmData[832].classification[0..3] := ' ';
   additionalAlarmData[833].classification[0..3] := ' ';
   additionalAlarmData[834].classification[0..3] := ' ';
   additionalAlarmData[835].classification[0..3] := ' ';
   additionalAlarmData[836].classification[0..3] := ' ';
   additionalAlarmData[837].classification[0..3] := ' ';
   additionalAlarmData[838].classification[0..3] := ' ';
   additionalAlarmData[839].classification[0..3] := ' ';
   additionalAlarmData[840].classification[0..3] := ' ';
   additionalAlarmData[841].classification[0..3] := ' ';
   additionalAlarmData[842].classification[0..3] := ' ';
   additionalAlarmData[843].classification[0..3] := ' ';
   additionalAlarmData[844].classification[0..3] := ' ';
   additionalAlarmData[845].classification[0..3] := ' ';
   additionalAlarmData[846].classification[0..3] := ' ';
   additionalAlarmData[847].classification[0..3] := ' ';
   additionalAlarmData[848].classification[0..3] := ' ';
   additionalAlarmData[849].classification[0..3] := ' ';
   additionalAlarmData[850].classification[0..3] := ' ';
   additionalAlarmData[851].classification[0..3] := ' ';
   additionalAlarmData[852].classification[0..3] := ' ';
   additionalAlarmData[853].classification[0..3] := ' ';
   additionalAlarmData[854].classification[0..3] := ' ';
   additionalAlarmData[855].classification[0..3] := ' ';
   additionalAlarmData[856].classification[0..3] := ' ';
   additionalAlarmData[857].classification[0..3] := ' ';
   additionalAlarmData[858].classification[0..3] := ' ';
   additionalAlarmData[859].classification[0..3] := ' ';
   additionalAlarmData[860].classification[0..3] := ' ';
   additionalAlarmData[861].classification[0..3] := ' ';
   additionalAlarmData[862].classification[0..3] := ' ';
   additionalAlarmData[863].classification[0..3] := ' ';
   additionalAlarmData[864].classification[0..3] := ' ';
   additionalAlarmData[865].classification[0..3] := ' ';
   additionalAlarmData[866].classification[0..3] := ' ';
   additionalAlarmData[867].classification[0..3] := ' ';
   additionalAlarmData[868].classification[0..3] := ' ';
   additionalAlarmData[869].classification[0..3] := ' ';
   additionalAlarmData[870].classification[0..3] := ' ';
   additionalAlarmData[871].classification[0..3] := ' ';
   additionalAlarmData[872].classification[0..3] := ' ';
   additionalAlarmData[873].classification[0..3] := ' ';
   additionalAlarmData[874].classification[0..3] := ' ';
   additionalAlarmData[875].classification[0..3] := ' ';
   additionalAlarmData[876].classification[0..3] := ' ';
   additionalAlarmData[877].classification[0..3] := ' ';
   additionalAlarmData[878].classification[0..3] := ' ';
   additionalAlarmData[879].classification[0..3] := ' ';
   additionalAlarmData[880].classification[0..3] := ' ';
   additionalAlarmData[881].classification[0..3] := ' ';
   additionalAlarmData[882].classification[0..3] := ' ';
   additionalAlarmData[883].classification[0..3] := ' ';
   additionalAlarmData[884].classification[0..3] := ' ';
   additionalAlarmData[885].classification[0..3] := ' ';
   additionalAlarmData[886].classification[0..3] := ' ';
   additionalAlarmData[887].classification[0..3] := ' ';
   additionalAlarmData[888].classification[0..3] := ' ';
   additionalAlarmData[889].classification[0..3] := ' ';
   additionalAlarmData[890].classification[0..3] := ' ';
   additionalAlarmData[891].classification[0..3] := ' ';
   additionalAlarmData[892].classification[0..3] := ' ';
   additionalAlarmData[893].classification[0..3] := ' ';
   additionalAlarmData[894].classification[0..3] := ' ';
   additionalAlarmData[895].classification[0..3] := ' ';
   additionalAlarmData[896].classification[0..3] := ' ';
   additionalAlarmData[897].classification[0..3] := ' ';
   additionalAlarmData[898].classification[0..3] := ' ';
   additionalAlarmData[899].classification[0..3] := ' ';
   additionalAlarmData[900].classification[0..3] := ' ';
   additionalAlarmData[901].classification[0..3] := ' ';
   additionalAlarmData[902].classification[0..3] := ' ';
   additionalAlarmData[903].classification[0..3] := ' ';
   additionalAlarmData[904].classification[0..3] := ' ';
   additionalAlarmData[905].classification[0..3] := ' ';
   additionalAlarmData[906].classification[0..3] := ' ';
   additionalAlarmData[907].classification[0..3] := ' ';
   additionalAlarmData[908].classification[0..3] := ' ';
   additionalAlarmData[909].classification[0..3] := ' ';
   additionalAlarmData[910].classification[0..3] := ' ';
   additionalAlarmData[911].classification[0..3] := ' ';
   additionalAlarmData[912].classification[0..3] := ' ';
   additionalAlarmData[913].classification[0..3] := ' ';
   additionalAlarmData[914].classification[0..3] := ' ';
   additionalAlarmData[915].classification[0..3] := ' ';
   additionalAlarmData[916].classification[0..3] := ' ';
   additionalAlarmData[917].classification[0..3] := ' ';
   additionalAlarmData[918].classification[0..3] := ' ';
   additionalAlarmData[919].classification[0..3] := ' ';
   additionalAlarmData[920].classification[0..3] := ' ';
   additionalAlarmData[921].classification[0..3] := ' ';
   additionalAlarmData[922].classification[0..3] := ' ';
   additionalAlarmData[923].classification[0..3] := ' ';
   additionalAlarmData[924].classification[0..3] := ' ';
   additionalAlarmData[925].classification[0..3] := ' ';
   additionalAlarmData[926].classification[0..3] := ' ';
   additionalAlarmData[927].classification[0..3] := ' ';
   additionalAlarmData[928].classification[0..3] := ' ';
   additionalAlarmData[929].classification[0..3] := ' ';
   additionalAlarmData[930].classification[0..3] := ' ';
   additionalAlarmData[931].classification[0..3] := ' ';
   additionalAlarmData[932].classification[0..3] := ' ';
   additionalAlarmData[933].classification[0..3] := ' ';
   additionalAlarmData[934].classification[0..3] := ' ';
   additionalAlarmData[935].classification[0..3] := ' ';
   additionalAlarmData[936].classification[0..3] := ' ';
   additionalAlarmData[937].classification[0..3] := ' ';
   additionalAlarmData[938].classification[0..3] := ' ';
   additionalAlarmData[939].classification[0..3] := ' ';
   additionalAlarmData[940].classification[0..3] := ' ';
   additionalAlarmData[941].classification[0..3] := ' ';
   additionalAlarmData[942].classification[0..3] := ' ';
   additionalAlarmData[943].classification[0..3] := ' ';
   additionalAlarmData[944].classification[0..3] := ' ';
   additionalAlarmData[945].classification[0..3] := ' ';
   additionalAlarmData[946].classification[0..3] := ' ';
   additionalAlarmData[947].classification[0..3] := ' ';
   additionalAlarmData[948].classification[0..3] := ' ';
   additionalAlarmData[949].classification[0..3] := ' ';
   additionalAlarmData[950].classification[0..3] := ' ';
   additionalAlarmData[951].classification[0..3] := ' ';
   additionalAlarmData[952].classification[0..3] := ' ';
   additionalAlarmData[953].classification[0..3] := ' ';
   additionalAlarmData[954].classification[0..3] := ' ';
   additionalAlarmData[955].classification[0..3] := ' ';
   additionalAlarmData[956].classification[0..3] := ' ';
   additionalAlarmData[957].classification[0..3] := ' ';
   additionalAlarmData[958].classification[0..3] := ' ';
   additionalAlarmData[959].classification[0..3] := ' ';
   additionalAlarmData[960].classification[0..3] := ' ';
   additionalAlarmData[961].classification[0..3] := ' ';
   additionalAlarmData[962].classification[0..3] := ' ';
   additionalAlarmData[963].classification[0..3] := ' ';
   additionalAlarmData[964].classification[0..3] := ' ';
